(* CODESYS project core.library
   Title: CW_Core
   Version: 0.3.0
   Placeholder: CW_Core
   Company: Climeworks AG

Project tree, tasks and I/O mapping:
  libraries: Tc2_Standard, * (Beckhoff Automation GmbH); Tc2_System, * (Beckhoff Automation GmbH); Tc2_Utilities, * (Beckhoff Automation GmbH); Tc3_Module, * (Beckhoff Automation GmbH); VisuDialogs, * (System)
  Clock/
    function block FB_Clock [ST]: end_of_day, ready, toString
    interface ITF_Clock: end_of_day, ready, toString
  i18n/
    data type E_Language
    function F_GetLanguageId [ST]
    function block FB_TextList [ST]: FB_init, get
    visualisation Frame_SwitchLanguage
    data type T_TranslatableName
    data type T_TranslatableText
  Implicit/
    function F_CheckRangeSigned [ST]
    function F_CheckRangeUnsigned [ST]
  Log/
    DataLogger/
      data type E_LoggerError
      function block FB_EventLoggableLogger [ST]: collectLog, FB_init, run
      function block FB_EventLogger [ST]: updateTimeFormat, useMilliseconds, _trigger, FB_init, trigger, triggerIf, triggerWithTime, write
      function block FB_ExternalTimestamp [ST]: end_of_day, ready, reset, setTime, toString
      function block FB_TimedLoggableLogger [ST]: collectLog, FB_init, run
      function block FB_TimedLogger [ST]: FB_init, write_sampled
      interface ITF_LogDataCollector: collectLog
      data type TIMESTAMPSTRING
    Interfaces/
      interface ITF_LogExtension: getLogTrigger
      interface ITF_Loggable: toLog
      interface ITF_Recordable: enableSelectionMode
    LogStack/
      data type E_LogSequence
      function block FB_LogStackManager [ST]: available, empty, getKey, getStackLevel, nextReadData, nextWritePtr, writeToStack, writeToStackData, writeToStackHeader
      function block FB_ResponseStackManager [ST]: getResponse, storeResponse
      interface ITF_WritableStack: available, getKey, writeToStackData, writeToStackHeader
      data type ST_logStackData
      data type ST_ResponseStack
    LogString/
      function block FB_LogString [ST]: logBoolProperty, logUdintProperty, logUintProperty, logBool, logReal, logString, logUdint, logUint, append, clear, concat, getLine, length, logAny, logValue, num_lines
      data type LOGSTRING
    LogWriter/
      function block FB_LogWriter [ST]: FB_init, full_filename, handleResponse, updateFileName, updateFileType, write
      data type ST_LogMessage
    data type E_LogMode
    global variables PL_Log
  ManualRecording/
    visualisation Frame_ManualRecording_display
    data type ST_Record
  Math/
    function F_NotZero [ST]
    function F_Ramp [ST]
  Mixin/
    Fallible/
      interface ITF_Fallible: get_name, has_error
    Pressure/
      data type E_PressureUnit
      function block FB_PressureMixin [ST]: bar, display_accuracy, from_mbar, mbar, pa
  Physics/
    SteamCondition/
      function F_P_SAT [ST]
      function F_T_SAT [ST]
    function F_sim_pressureFlow [ST]
  StringSizes/
    data type NAME_STRING
    global variables PL_StringSizes
    data type TAG_STRING
  TEST/
    lib/
      function block FB_Test [ST]: check
      program TEST_TEMPLATE [ST]
    Utils/
      program TEST_BITS [ST]
      program TEST_TIMESTRUCT_INCREMENT [ST]: assertEqual
    program TEST [ST]
  Utils/
    Bits/
      function SET_BIT_IN_BYTE [ST]
      function SET_BIT_IN_BYTE_ARRAY [ST]
    Endian/
      function F_IntSwapEndian [ST]
      function F_SafeRealSwapEndian [ST]
      function F_SafeRealSwapWords [ST]
      data type Float32
      data type Int16
    Limits/
      Visu/
        visualisation Frame_IntLimits
        visualisation Frame_RealLimits
        visualisation Frame_UdintLimits
        visualisation Frame_UsintLimits
        text list TL_DisplayAccuracy
      data type ST_BaseLimits
      data type ST_DintLimits
      data type ST_IntLimits
      data type ST_RealLimits
      data type ST_UdintLimits
      data type ST_UintLimits
      data type ST_UsintLimits
    String/
      Concat/
        function CONCAT3 [ST]
        function CONCAT4 [ST]
        function CONCAT5 [ST]
        function CONCAT6 [ST]
      Placeholder/
        function F_ResolvePlaceholder [ST]
        data type PLACEHOLDER_STRING
      function F_FindAndReplace [ST]
      function F_FindAndReplaceAll [ST]
      function F_Glue [ST]
      function F_ReplaceX [ST]
      function FILL_WIDTH [ST]
    Ternary/
      function BOOL_TO_TERNARY [ST]
      data type E_Ternary
    Time/
      data type E_TIME_UNIT
      function block FB_Blinker [ST]
      function block FB_TimeDelta [ST]: reset
      function block FB_TON_PAUSABLE [ST]
      function SYSTEMTIME_TO_STRING [ST]
      function TIME_TO_FSTRING [ST]
      function TIMESTRUCT_INCREMENT [ST]
    function block FB_RememberRestore [ST]: remember, restore
    function block FB_ResourceManager [ST]: available, FB_init, release, reserve
*)

// i18n/E_Language
{attribute 'qualified_only'}
TYPE E_Language :
(
	de := 0,
	en,
	num
)UINT;
END_TYPE

// i18n/T_TranslatableName
TYPE T_TranslatableName : ARRAY[0..E_Language.num-1] OF NAME_STRING; END_TYPE

// i18n/T_TranslatableText
TYPE T_TranslatableText : ARRAY[0..E_Language.num-1] OF T_MaxString; END_TYPE

// Log/DataLogger/E_LoggerError
{attribute 'qualified_only'}
{attribute 'strict'}
TYPE E_LoggerError :
(
	ok := 0,
	trigger_overflow
) UDINT;
END_TYPE

// Log/DataLogger/TIMESTAMPSTRING
TYPE TIMESTAMPSTRING : STRING(30); END_TYPE

// Log/LogStack/E_LogSequence
{attribute 'qualified_only'}
{attribute 'strict'}
TYPE E_LogSequence :
(
	daily		:= 1,
	weekly		:= 2,
	monthly		:= 4,
	yearly		:= 8,
	perCycle	:= 16,
	unlimited	:= 32,
	other1		:= 64,
	other2		:= 128
) WORD;
END_TYPE

// Log/LogStack/ST_logStackData
TYPE ST_logStackData :
STRUCT
	type_of_data : INT;			// 0: data	1:Header
	key : INT;					// Response: Key ID
	file_name : STRING[64];		// C# Len=65		 = “Betriebsdaten.log”
	file_type : WORD;			// FileType          = 01h (=daily)
								// 1: daily
								// 2: weekly
								// 4: monthly
								// 8: yearly
								// 16: per cycle
								// 32: unlimited
								// 64: other features (example: overwrite file on restart)
								// 128: other features
	cycle : INT;				// Process Cycle when fileType 16 is used
	option : INT;
	header_or_data : STRING[255]; // C# Len=256
	eom : BOOL;					// End of Message
END_STRUCT
END_TYPE

// Log/LogStack/ST_ResponseStack
TYPE ST_ResponseStack :
STRUCT
	// Response
	key			:INT;			// Response: Key ID
	fault_code	:INT;			// NONE 				= 0	V1.00-X31
        						// KEY 					= 1 // Key ist dem Feurer-Tool nicht mehr bekannt. Vermutlich wurde es neugestartet. Header muss erneut gesendet werden.
        						// FILE_MISSING 		= 2
        						// FILENAME_MISSING 	= 3
        						// FILESYSTEM 			= 4 // Wahrscheinlich Speicher voll?
        						// SERIALIZATION 		= 5
        						// NULLMSG 				= 99
	error		:BOOL;			// Response: Error
END_STRUCT
END_TYPE

// Log/LogString/LOGSTRING
TYPE LOGSTRING : ARRAY[1..PL_Log.max_lines] OF STRING(255); END_TYPE

// Log/LogWriter/ST_LogMessage
TYPE ST_LogMessage :
STRUCT
	header	: FB_LogString := ( get_header := TRUE, force_get_data := TRUE );
	data	: FB_LogString;
END_STRUCT
END_TYPE

// Log/E_LogMode
{attribute 'qualified_only'}
TYPE E_LogMode :
(
	no := 0,
	yes,
	on_change
);
END_TYPE

// ManualRecording/ST_Record
TYPE ST_Record :
STRUCT
	enabled : BOOL;  // if true, this will be recorded in the manual recording
	selection_mode : BOOL;  // if true, this should show an option on the HMI to be selected for recording
END_STRUCT
END_TYPE

// Mixin/Pressure/E_PressureUnit
{attribute 'qualified_only'}
{attribute 'strict'}
TYPE E_PressureUnit :
(
	mbar := 0,
	bar,
	pa
);
END_TYPE

// StringSizes/NAME_STRING
TYPE NAME_STRING : STRING(PL_StringSizes.name_string_size); END_TYPE

// StringSizes/TAG_STRING
TYPE TAG_STRING : STRING(PL_StringSizes.tag_string_size); END_TYPE

// Utils/Endian/Float32
TYPE Float32 :
UNION
	float : REAL;
	dword_ : DWORD;
	words : ARRAY[0..1] OF WORD;
	bytes : ARRAY[0..3] OF BYTE;
END_UNION
END_TYPE

// Utils/Endian/Int16
TYPE Int16 :
UNION
	uinteger : UINT;
	integer : INT;
	bytes : ARRAY[0..1] OF BYTE;
END_UNION
END_TYPE

// Utils/Limits/ST_BaseLimits
TYPE ST_BaseLimits :
STRUCT
	display_font_size : UINT(0..40) := 9;  //pt
END_STRUCT
END_TYPE

// Utils/Limits/ST_DintLimits
TYPE ST_DintLimits EXTENDS ST_BaseLimits :
STRUCT
	low : DINT;
	high : DINT;
END_STRUCT
END_TYPE

// Utils/Limits/ST_IntLimits
TYPE ST_IntLimits EXTENDS ST_BaseLimits :
STRUCT
	low : INT;
	high : INT;
END_STRUCT
END_TYPE

// Utils/Limits/ST_RealLimits
TYPE ST_RealLimits EXTENDS ST_BaseLimits :
STRUCT
	low : REAL;
	high : REAL;
	display_accuracy : UINT(0..4) := 1;
END_STRUCT
END_TYPE

// Utils/Limits/ST_UdintLimits
TYPE ST_UdintLimits EXTENDS ST_BaseLimits:
STRUCT
	low : UDINT;
	high : UDINT;
END_STRUCT
END_TYPE

// Utils/Limits/ST_UintLimits
TYPE ST_UintLimits EXTENDS ST_BaseLimits :
STRUCT
	low : UINT;
	high : UINT;
END_STRUCT
END_TYPE

// Utils/Limits/ST_UsintLimits
TYPE ST_UsintLimits EXTENDS ST_BaseLimits :
STRUCT
	low : USINT;
	high : USINT;
END_STRUCT
END_TYPE

// Utils/String/Placeholder/PLACEHOLDER_STRING
TYPE PLACEHOLDER_STRING : STRING(3); END_TYPE

// Utils/Ternary/E_Ternary
{attribute 'qualified_only'}
{attribute 'strict'}
TYPE E_Ternary :
(
	unset := 0,
	yes,
	no
)USINT;
END_TYPE

// Utils/Time/E_TIME_UNIT
{attribute 'qualified_only'}
{attribute 'strict'}
TYPE E_TIME_UNIT :
(
	millisecond := 0,
	second,
	minute,
	hour,
	day
);
END_TYPE

// Log/PL_Log
{attribute 'qualified_only'}
VAR_GLOBAL CONSTANT
	max_lines : INT := 65;  // size of FB_LogString
	log_stack_size : INT := 90;  // size of Log Stack (should be bigger than log string)
END_VAR

// StringSizes/PL_StringSizes
{attribute 'qualified_only'}
VAR_GLOBAL CONSTANT
	name_string_size : UINT := 40;
	tag_string_size : UINT := 15;
END_VAR

// Clock/FB_Clock
FUNCTION_BLOCK FB_Clock IMPLEMENTS ITF_Clock
VAR_OUTPUT
	date_time_initialized	: BOOL; // TRUE, sobald dateTime korrekten Wert enthält
	date_time				: TIMESTRUCT; // Aktuelle Datumzeit des Systems
	end_of_year				: BOOL; // TRUE bei Jahreswechsel
	end_of_month			: BOOL; // TRUE bei Monatswechsel
	_end_of_day				: BOOL; // TRUE bei Tageswechsel
END_VAR
VAR
	nt_get_time				: NT_GetTime;
END_VAR
VAR PERSISTENT
	last_date_time			: TIMESTRUCT; // Zeit des letzten Zyklus
END_VAR

// Datum und Uhrzeit in einen Timestruct schreiben
nt_get_time(START:=TRUE, TIMESTR=>date_time);
IF NOT nt_get_time.BUSY THEN
	date_time_initialized := TRUE;
	nt_get_time(START:=FALSE); // Zurücksetzen
ELSIF date_time_initialized THEN
	// increment time while nt_get_time is busy to prevent duplicate timestamp in logs
	date_time := TIMESTRUCT_INCREMENT( date_time, UDINT_TO_UINT(TwinCAT_SystemInfoVarList._TaskInfo[GETCURTASKINDEXEX()].CycleTime/10000) );
END_IF

// Sobald Systemzeit gelesen wurde..
IF date_time_initialized THEN

	// Jahreswechsel detektieren
	IF (date_time.wYear > last_date_time.wYear) THEN
		end_of_year := TRUE;
	ELSE
		end_of_year := FALSE;
	END_IF

	// Monatswechsel detektieren
	IF (date_time.wMonth > last_date_time.wMonth) AND date_time.wYear = last_date_time.wYear OR (date_time.wYear > last_date_time.wYear) THEN
		end_of_month := TRUE;
	ELSE
		end_of_month := FALSE;
	END_IF

	// Mitternacht detektieren
	IF (date_time.wDay > last_date_time.wDay) AND date_time.wMonth = last_date_time.wMonth OR (date_time.wMonth > last_date_time.wMonth) THEN
		_end_of_day := TRUE;
	ELSE
		_end_of_day := FALSE;
	END_IF

	// Letztes Datum merken
	last_date_time	:= date_time;
END_IF

PROPERTY end_of_day : BOOL
GET
end_of_day := _end_of_day;
END_GET
END_PROPERTY

PROPERTY ready : BOOL
// returns true, if clock is ready for use
GET
ready := date_time_initialized;
END_GET
END_PROPERTY

METHOD toString : STRING
VAR_INPUT
	format		: STRING;
END_VAR
toString := SYSTEMTIME_TO_STRING( date_time, format );
END_METHOD

END_FUNCTION_BLOCK

// Utils/Time/TIMESTRUCT_INCREMENT
FUNCTION TIMESTRUCT_INCREMENT : TIMESTRUCT
VAR_INPUT
	base : TIMESTRUCT;
	increment : UINT;  // in ms
END_VAR

// increases the timestruct by increment
IF	base.wMilliseconds + increment < 1000 THEN
	TIMESTRUCT_INCREMENT := base;
	TIMESTRUCT_INCREMENT.wMilliseconds := base.wMilliseconds + increment;
ELSE
	// DT looses milliseconds (rounded)
	TIMESTRUCT_INCREMENT := base;
	TIMESTRUCT_INCREMENT.wMilliseconds := 0;
	TIMESTRUCT_INCREMENT := DT_TO_SYSTEMTIME(SYSTEMTIME_TO_DT(TIMESTRUCT_INCREMENT) + UINT_TO_TIME((base.wMilliseconds + increment)/1000*1000));
	TIMESTRUCT_INCREMENT.wMilliseconds := ( base.wMilliseconds + increment ) MOD 1000;
END_IF

END_FUNCTION

// Clock/ITF_Clock
INTERFACE ITF_Clock

PROPERTY end_of_day : BOOL
GET
END_GET
END_PROPERTY

PROPERTY ready : BOOL
// returns true, if clock is ready for use
GET
END_GET
END_PROPERTY

METHOD toString : STRING
VAR_INPUT
	format		: STRING;
END_VAR
END_METHOD

END_INTERFACE

// Utils/Time/SYSTEMTIME_TO_STRING
FUNCTION SYSTEMTIME_TO_STRING : STRING
VAR_INPUT
	system_time	: TIMESTRUCT;
	format		: STRING;
END_VAR
VAR
	tmp_string	: STRING;
END_VAR

SYSTEMTIME_TO_STRING := format;

// aktuelle Zeit (%T)
SYSTEMTIME_TO_STRING := F_FindAndReplace( SYSTEMTIME_TO_STRING, '%T', '%H:%M:%S' );


// Jahr 4-Stellig
IF system_time.wYear < 10 THEN
	tmp_string := CONCAT ('0', WORD_TO_STRING(system_time.wYear));
ELSE
	tmp_string := WORD_TO_STRING(system_time.wYear);
END_IF
SYSTEMTIME_TO_STRING := F_FindAndReplace( SYSTEMTIME_TO_STRING, '%Y', tmp_string );


// Monat
IF system_time.wMonth < 10 THEN
	tmp_string := CONCAT ('0', WORD_TO_STRING(system_time.wMonth));
ELSE
	tmp_string := WORD_TO_STRING(system_time.wMonth);
END_IF
SYSTEMTIME_TO_STRING := F_FindAndReplace( SYSTEMTIME_TO_STRING, '%m', tmp_string );


// Tag des Monats
IF system_time.wDay < 10 THEN
	tmp_string := CONCAT ('0', WORD_TO_STRING(system_time.wDay));
ELSE
	tmp_string := WORD_TO_STRING(system_time.wDay);
END_IF
SYSTEMTIME_TO_STRING := F_FindAndReplace( SYSTEMTIME_TO_STRING, '%d', tmp_string );


// h (%H) (Bereich 00 bis 23)
IF system_time.wHour < 10 THEN
	tmp_string := CONCAT ('0', WORD_TO_STRING(system_time.wHour));
ELSE
	tmp_string := WORD_TO_STRING(system_time.wHour);
END_IF
SYSTEMTIME_TO_STRING := F_FindAndReplace( SYSTEMTIME_TO_STRING, '%H', tmp_string );

// min (%M) (Bereich 00 bis 59)
IF system_time.wMinute < 10 THEN
	tmp_string := CONCAT ('0', WORD_TO_STRING(system_time.wMinute));
ELSE
	tmp_string := WORD_TO_STRING(system_time.wMinute);
END_IF
SYSTEMTIME_TO_STRING := F_FindAndReplace( SYSTEMTIME_TO_STRING, '%M', tmp_string );

// sec (%S)
IF system_time.wSecond < 10 THEN
	tmp_string := CONCAT ('0', WORD_TO_STRING(system_time.wSecond));
ELSE
	tmp_string := WORD_TO_STRING(system_time.wSecond);
END_IF
SYSTEMTIME_TO_STRING := F_FindAndReplace( SYSTEMTIME_TO_STRING, '%S', tmp_string );

// Millisec (%f)
IF system_time.wMilliseconds < 10 THEN
	tmp_string := CONCAT ('00', WORD_TO_STRING(system_time.wMilliseconds));
ELSIF system_time.wMilliseconds < 100 THEN
	tmp_string := CONCAT ('0', WORD_TO_STRING(system_time.wMilliseconds));
ELSE
	tmp_string := WORD_TO_STRING(system_time.wMilliseconds);
END_IF
SYSTEMTIME_TO_STRING := F_FindAndReplace( SYSTEMTIME_TO_STRING, '%f', tmp_string );

END_FUNCTION

// Utils/String/F_FindAndReplace
FUNCTION F_FindAndReplace : STRING
VAR_INPUT
	str : T_MaxString;
	find_str : T_MaxString;
	replace_str : T_MaxString;
END_VAR
VAR_OUTPUT
	found : BOOL; 
END_VAR
VAR
	p : INT;
END_VAR

p := FIND( str, find_str );
found := p > 0;
IF found THEN
	F_FindAndReplace := REPLACE( str, replace_str, LEN(find_str), p );
ELSE
	F_FindAndReplace := str;
END_IF

END_FUNCTION

// i18n/F_GetLanguageId
FUNCTION F_GetLanguageId : E_Language
// Gibt die aktuelle Sprache der Visu zurück
VAR_INPUT
END_VAR
VAR
	language : STRING;
END_VAR

language := VisuElems.cmpDynamictext.DynamicTextGetCurrentLanguage();
IF language = '' OR language = 'default' OR language = 'de' THEN
	F_GetLanguageId := E_Language.de;
ELSE
	F_GetLanguageId := E_Language.en;
END_IF

END_FUNCTION

// i18n/FB_TextList
FUNCTION_BLOCK FB_TextList
VAR_INPUT
END_VAR
VAR_OUTPUT
END_VAR
VAR
	text_list_path : STRING;
END_VAR

METHOD FB_init : BOOL
VAR_INPUT
	bInitRetains : BOOL; // if TRUE, the retain variables are initialized (warm start / cold start)
	bInCopyCode   : BOOL;  // if TRUE, the instance afterwards gets moved into the copy code (online change)
	text_list : STRING;
END_VAR
text_list_path := text_list;
END_METHOD

METHOD get : STRING
VAR_INPUT
	index : UINT;
END_VAR
VAR
	language : STRING;
	index_string : STRING;
END_VAR
index_string := UINT_TO_STRING(index);

language := VisuElems.cmpDynamictext.DynamicTextGetCurrentLanguage();
IF language = '' OR language = 'default' THEN
	get := VisuElems.cmpDynamictext.DynamicTextGetDefaultText(ADR(text_list_path), ADR(index_string))^;
ELSE
	get := VisuElems.cmpDynamictext.DynamicTextGetText(ADR(text_list_path), ADR(index_string))^;
END_IF
END_METHOD

END_FUNCTION_BLOCK

// Implicit/F_CheckRangeSigned
// Implicitly generated code : DO NOT EDIT
FUNCTION F_CheckRangeSigned : DINT
VAR_INPUT
	value, lower, upper: DINT;
END_VAR

// Implicitly generated code : Only an Implementation suggestion
{noflow}
IF (value < lower) THEN
	F_CheckRangeSigned := lower;
ELSIF(value > upper) THEN
	F_CheckRangeSigned := upper;
ELSE
	F_CheckRangeSigned := value;
END_IF
{flow}

END_FUNCTION

// Implicit/F_CheckRangeUnsigned
// Implicitly generated code : DO NOT EDIT
FUNCTION F_CheckRangeUnsigned : UDINT
VAR_INPUT
	value, lower, upper: UDINT;
END_VAR

// Implicitly generated code : Only an Implementation suggestion
{noflow}
IF (value < lower) THEN
	F_CheckRangeUnsigned := lower;
ELSIF(value > upper) THEN
	F_CheckRangeUnsigned := upper;
ELSE
	F_CheckRangeUnsigned := value;
END_IF
{flow}

END_FUNCTION

// Log/DataLogger/FB_EventLoggableLogger
FUNCTION_BLOCK FB_EventLoggableLogger EXTENDS FB_EventLogger IMPLEMENTS ITF_LogDataCollector
VAR
	// loggable to get data from
	loggable : ITF_Loggable;

	// settings
	log_type : UINT;
END_VAR

METHOD collectLog : BOOL
VAR_IN_OUT
	log_string	: FB_LogString;
END_VAR
VAR_INPUT
	timestamp : TIMESTAMPSTRING;  // is "Time;" for header and current timestamp + ';' as string for data
END_VAR
log_string.append(timestamp);
loggable.toLog( log_string, log_type );
END_METHOD

METHOD FB_init : BOOL
VAR_INPUT
	bInitRetains : BOOL; // if TRUE, the retain variables are initialized (warm start / cold start)
	bInCopyCode : BOOL;  // if TRUE, the instance afterwards gets moved into the copy code (online change)
	file_name	: STRING(53);
END_VAR
log_writer.updateFileName(file_name);
END_METHOD

METHOD run : BOOL
VAR_INPUT
	loggable : ITF_Loggable;
	stack : ITF_WritableStack;
	clock : ITF_Clock;
	file_writer_connected : BOOL;
END_VAR
// Den loggable für die collect-Methoden erreichbar machen
THIS^.loggable := loggable;
// Logger laufen lassen.
write( data_collector := THIS^, stack, file_writer_connected );
END_METHOD

END_FUNCTION_BLOCK

// Log/DataLogger/FB_EventLogger
FUNCTION_BLOCK FB_EventLogger;
VAR_INPUT
	force_get_data : BOOL; //TRUE: force the values of all elements to be appended to the log_string, FALSE: elements decide if append the data or not
END_VAR
VAR_OUTPUT
	error : BOOL;
	error_id : UDINT;
	last_timestamp : TIMESTAMPSTRING;  // last timestamp of an internal trigger to be used to inform external triggers
END_VAR
VAR_INPUT
	max_triggering_interval : USINT := 3; // Maximum interval between consecutive triggering (i.e. lines in the log file). Unit is program cycles
END_VAR
VAR
	message : ST_LogMessage;
	header_cached : BOOL;  // TRUE, wenn header gecached wurde
	// triggering
	triggered : BOOL; // TRUE: event logger has been triggered, FALSE: event logger is not being triggered

	// writer
	log_writer : FB_LogWriter('EventLogger', E_LogSequence.daily);
	data_collected : BOOL; // TRUE: data has been collected

	// timestamp settings
	time_header : TIMESTAMPSTRING := 'Time;';
	time_format : STRING := '%Y-%m-%d %H:%M:%S';
	timestamp : TIMESTAMPSTRING;
END_VAR

METHOD updateTimeFormat : BOOL
VAR_INPUT
	new_time_format : STRING;
END_VAR
time_format := new_time_format;
END_METHOD

METHOD useMilliseconds : BOOL
VAR_INPUT
	use_milliseconds : BOOL;
END_VAR
IF use_milliseconds THEN
	time_format := CONCAT( time_format, '.%f' );
END_IF
END_METHOD

// basic trigger
METHOD PRIVATE _trigger : BOOL
VAR_INPUT
	clock : ITF_Clock;
END_VAR
{warning 'the clock may not be ready here. check somewhere else'}
timestamp := clock.toString(time_format);
triggered := TRUE;
END_METHOD

METHOD FB_init : BOOL
VAR_INPUT
	bInitRetains : BOOL; // if TRUE, the retain variables are initialized (warm start / cold start)
	bInCopyCode : BOOL;  // if TRUE, the instance afterwards gets moved into the copy code (online change)
END_VAR
log_writer.updateFileType(E_LogSequence.daily);  // legacy default.
END_METHOD

// trigger for module internal triggering with own timestamp
METHOD trigger : BOOL
VAR_INPUT
	clock : ITF_Clock;
END_VAR
{warning 'the clock may not be ready here. check somewhere else'}
_trigger(clock);
last_timestamp := timestamp;  // remember for external trigger
END_METHOD

METHOD triggerIf : BOOL
VAR_INPUT
	condition : BOOL;
	clock : ITF_Clock;
END_VAR
IF condition THEN
	trigger(clock);
END_IF
triggerIf := triggered;
END_METHOD

// trigger for external triggering with other timestamp
METHOD triggerWithTime : BOOL
VAR_INPUT
	external_timestamp : REFERENCE TO FB_ExternalTimestamp;
END_VAR
IF external_timestamp.triggered THEN
	_trigger(external_timestamp);
END_IF
END_METHOD

METHOD write : BOOL
VAR_INPUT
	data_collector : ITF_LogDataCollector;
	stack : ITF_WritableStack;
	file_writer_connected : BOOL;
END_VAR
VAR_INST
	write_to_log : BOOL;
	consecutive_trigger_counter : USINT;
END_VAR
// 1. Header zusammensetzen und senden
IF NOT header_cached THEN
	message.header.clear();
	data_collector.collectLog( message.header, time_header );
	header_cached := TRUE;
	write_to_log := TRUE;
END_IF

// 2. If log_writer has not been initialized, i.e. header has not been written, force get a complete log_string of data (second line after header should always been complete).
IF NOT log_writer.status_initialized THEN
	message.data.force_get_data := TRUE;
ELSE
	message.data.force_get_data := force_get_data;
END_IF

// Trigger overflow watchdog
IF triggered THEN
	consecutive_trigger_counter := consecutive_trigger_counter + 1;

	IF consecutive_trigger_counter > max_triggering_interval THEN
		error := TRUE;
		error_id := E_LoggerError.trigger_overflow;
		consecutive_trigger_counter := 0;
		data_collected := FALSE;
	END_IF
ELSE
	error := FALSE;
	consecutive_trigger_counter := 0;
	data_collected := FALSE;
END_IF

// 2. Daten zusammensetzen
IF triggered AND NOT data_collected THEN
	message.data.clear();
	data_collector.collectLog( message.data, CONCAT(timestamp, ';') );
	data_collected := TRUE; // reset
END_IF
triggered := FALSE;

// 4. Header und/oder Daten schreiben
// TODO: Auslesen, ob ein Fehler aufgetreten ist #SafetyChecks
// IMPORTANT: this write method must be called regularly, to resend the header if pydialogs restarted
IF log_writer.write(message, stack, file_writer_connected) THEN
	message.data.clear();
END_IF

// Reset Error ID
IF NOT error THEN
	error_id := E_LoggerError.ok;
END_IF
END_METHOD

END_FUNCTION_BLOCK

// Log/LogWriter/FB_LogWriter
FUNCTION_BLOCK FB_LogWriter
VAR_INPUT
	cycle : INT;  // Process Cycle when fileType "perCycle" is used
END_VAR
VAR_OUTPUT
	// TODO: Bei error könnte eine Warnung auslösen.
	error_response :BOOL;
	fault_code :INT;			// NONE 				= 0	V1.00-X31
        						// KEY 					= 1 // Key ist dem Feurer-Tool nicht mehr bekannt. Vermutlich wurde es neugestartet. Header muss erneut gesendet werden.
        						// FILE_MISSING 		= 2
        						// FILENAME_MISSING 	= 3
        						// FILESYSTEM 			= 4 // Wahrscheinlich Speicher voll?
        						// SERIALIZATION 		= 5
        						// NULLMSG 				= 99
	error_full_stack : BOOL;
	status_initialized : BOOL := FALSE;
END_VAR
VAR
	// settings
	key : INT;  // Response: Key ID
	file_prefix : STRING(20);
	file_extension : STRING(10) := 'csv';
	file_name : STRING(60);  // Dateiname ohne Endung
	file_type : E_LogSequence;  // FileType

	//
	//stack_manager : REFERENCE TO FB_LogStackManager;
END_VAR

METHOD FB_init : BOOL
VAR_INPUT
	bInitRetains : BOOL; // if TRUE, the retain variables are initialized (warm start / cold start)
	bInCopyCode : BOOL;  // if TRUE, the instance afterwards gets moved into the copy code (online change)
	file_name	: STRING(53);
	file_type	: E_LogSequence; // FileType
END_VAR
THIS^.file_name := file_name;
THIS^.file_type := file_type;
END_METHOD

PROPERTY full_filename : STRING(100)
GET
IF file_prefix <> '' THEN
	full_filename := CONCAT5(file_prefix, '_', file_name, '.', file_extension);
ELSE
	full_filename := CONCAT3(file_name, '.', file_extension);
END_IF
END_GET
END_PROPERTY

METHOD handleResponse : BOOL
VAR_INPUT
	response : ST_ResponseStack;
END_VAR
error_response := response.error;
fault_code := response.fault_code;
END_METHOD

METHOD updateFileName : BOOL
VAR_INPUT
	new_file_name : STRING(60);
END_VAR
file_name := new_file_name;
status_initialized := FALSE; // Muss neu initialisiert werden.
END_METHOD

METHOD updateFileType : BOOL
VAR_INPUT
	new_file_type : E_LogSequence;
END_VAR
file_type := new_file_type;
status_initialized := FALSE; // Muss neu initialisiert werden.
END_METHOD

METHOD write : BOOL
VAR_IN_OUT
	message	: ST_LogMessage;
END_VAR
VAR_INPUT
	stack_manager : ITF_WritableStack;
	file_writer_connected : BOOL;
END_VAR
VAR
	i : UINT;
END_VAR
VAR_INST
	initialized: BOOL;
END_VAR
// get key the first time
IF NOT initialized THEN
	key := stack_manager.getKey();
	initialized := TRUE;
END_IF

// Filing anhalten, wenn Dialogs nicht verbunden ist.
IF NOT file_writer_connected THEN
	status_initialized := FALSE; // Header muss erneut geschrieben werden, wenn Verbindung wieder aufgebaut wurde.
	RETURN;
END_IF

// Header nach Fehler erneut senden.
IF error_response OR fault_code <> 0 THEN
	status_initialized := FALSE;
END_IF

// Header
IF NOT status_initialized AND message.header.length > 0 AND stack_manager.available >= message.header.num_lines THEN
	// Setup & Init
	FOR i:=1 TO message.header.num_lines DO
		// Teil i Header in den Stack schreiben
		error_full_stack := NOT stack_manager.writeToStackHeader (
			key := key,
			file_name := full_filename,
			file_type := file_type,  // FileType
			cycle := cycle,  // Process Cycle when fileType 16 is used
			option := 0,
			header := message.header.getLine(i),  // C# Len=256
			eom := (i=message.header.num_lines)  // End of Message
		);
	END_FOR
	status_initialized:=TRUE;
END_IF

// Data
IF status_initialized AND message.data.length > 0 AND stack_manager.available >= message.data.num_lines THEN
	FOR i:=1 TO message.data.num_lines DO
		// Hier werden die Daten in den Stack geschrieben
		error_full_stack := NOT stack_manager.writeToStackData(
			key := key,
			data := message.data.getLine(i),
			eom := (i=message.data.num_lines)  // End of Message
		);
	END_FOR
	write := TRUE;
END_IF
END_METHOD

END_FUNCTION_BLOCK

// Log/LogStack/FB_LogStackManager
{attribute 'analysis' := '-2'} // yes this is empty
FUNCTION_BLOCK FB_LogStackManager IMPLEMENTS ITF_WritableStack
VAR
	log_stack_read				:INT := 0;
	log_stack_write				:INT := 0;
	log_stack_data				:ARRAY[0..PL_Log.log_stack_size-1] OF ST_logStackData;
	stack_full					:BOOL;
	//log_stack_sent, log_stack_received :ARRAY[0..log_stack_size-1] OF BOOL;
	
	next_key : INT;
END_VAR

PROPERTY available : UINT
GET
available := INT_TO_UINT(( log_stack_read - log_stack_write - 1 + PL_Log.log_stack_size ) MOD PL_Log.log_stack_size);
END_GET
END_PROPERTY

PROPERTY empty : BOOL
GET
empty := log_stack_read = log_stack_write;
END_GET
END_PROPERTY

METHOD getKey : INT;
// Do not call this method in declaration part of in FB_init
getKey := next_key;
next_key := next_key + 1;
END_METHOD

METHOD getStackLevel : REAL
VAR_INPUT
END_VAR
getStackLevel := INT_TO_REAL( ( log_stack_write - log_stack_read + PL_Log.log_stack_size ) MOD PL_Log.log_stack_size ) / PL_Log.log_stack_size;
END_METHOD

METHOD nextReadData : ST_logStackData // Gibt Referenz auf nächte zu lesende Zeile zurück.
VAR_INPUT
END_VAR
log_stack_read := (log_stack_read + 1) MOD PL_Log.log_stack_size;
nextReadData := log_stack_data[log_stack_read];
END_METHOD

METHOD PRIVATE nextWritePtr : POINTER TO ST_logStackData // Gibt Pointer auf nächte zu lesende Zeile zurück.
VAR_INPUT
END_VAR
VAR
	tmp : INT;
END_VAR
tmp := (log_stack_write + 1) MOD PL_Log.log_stack_size;

// Wenn Stack voll ist, keine Referenz zurückgeben. Write-Pointer bleibt unverändert.
IF stack_full := tmp = log_stack_read THEN
	nextWritePtr := 0;
	//Setze EOM beim letzen Eintrag
	log_stack_data[log_stack_write].eom := TRUE;
	RETURN;
END_IF
log_stack_write := tmp;

nextWritePtr := ADR(log_stack_data[log_stack_write]);
END_METHOD

METHOD PRIVATE writeToStack : BOOL // Gibt True zurück, wenn In Stack geschrieben werden konnte.
VAR_INPUT
	type_of_data		:INT;			// Header = 0, Data = 1
	key			:INT;			// Response: Key ID
	file_name 		:STRING[64];	// C# Len=65		 = “Betriebsdaten.log”
	file_type		:WORD;			// FileType          = 01h (=daily)
	cycle			:INT;			// Process Cycle when fileType 16 is used
	option			:INT;
	header_or_data	:STRING[255];	// C# Len=256
	eom				:BOOL;			// End of Message
END_VAR
VAR
	write		: POINTER TO ST_logStackData;
END_VAR
write := nextWritePtr();
IF write <> 0 THEN
	write^.type_of_data := type_of_data;
	write^.key := key;
	write^.file_name := file_name;
	write^.file_type := file_type;

	write^.cycle := cycle;
	write^.option := option;
	write^.header_or_data := header_or_data;
	write^.eom := eom;
	writeToStack := TRUE; // Return TRUE
END_IF;
END_METHOD

METHOD writeToStackData : BOOL
VAR_INPUT
	key :INT;			// Response: Key ID
	data :STRING[255];	// C# Len=256
	eom :BOOL;			// End of Message
END_VAR
VAR
	success			: BOOL;
END_VAR
success := writeToStack(
	type_of_data := 1,  // Explizit data
	key := key,
	file_name := '',
	file_type := 0,
	cycle := 0,
	option := 0,
	header_or_data := data,
	eom := eom
);

writeToStackData := success;
END_METHOD

METHOD writeToStackHeader : BOOL
VAR_INPUT
	key			: INT;			// Response: Key ID
	file_name 	: STRING[64];	// C# Len=65		 = “Betriebsdaten.log”
	file_type	: E_LogSequence;	// FileType
	cycle		: INT;			// Process Cycle when fileType 16 is used
	option		: INT;
	header		: STRING[255];	// C# Len=256
	eom			: BOOL;			// End of Message
END_VAR
VAR
	success		: BOOL;
END_VAR
success := writeToStack(
	type_of_data := 0, // Explizit header
	key := key,
	file_name := file_name,
	file_type := file_type,
	cycle := cycle,
	option := option,
	header_or_data := header,
	eom := eom
);

writeToStackHeader := success;
END_METHOD

END_FUNCTION_BLOCK

// Log/LogStack/ITF_WritableStack
INTERFACE ITF_WritableStack

PROPERTY available : UINT
GET
END_GET
END_PROPERTY

METHOD getKey : INT;
END_METHOD

METHOD writeToStackData : BOOL
VAR_INPUT
	key :INT;			// Response: Key ID
	data :STRING[255];	// C# Len=256
	eom :BOOL;			// End of Message
END_VAR
END_METHOD

METHOD writeToStackHeader : BOOL
VAR_INPUT
	key			: INT;			// Response: Key ID
	file_name 	: STRING[64];	// C# Len=65		 = “Betriebsdaten.log”
	file_type	: E_LogSequence;	// FileType
	cycle		: INT;			// Process Cycle when fileType 16 is used
	option		: INT;
	header		: STRING[255];	// C# Len=256
	eom			: BOOL;			// End of Message
END_VAR
END_METHOD

END_INTERFACE

// Utils/String/Concat/CONCAT5
FUNCTION CONCAT5 : T_MaxString
VAR_INPUT
	string1 : T_MaxString;
	string2 : T_MaxString;
	string3 : T_MaxString;
	string4 : T_MaxString;
	string5 : T_MaxString;
END_VAR
VAR
END_VAR

CONCAT5 := CONCAT( CONCAT( CONCAT ( CONCAT ( string1, string2 ), string3) , string4 ), string5 );

END_FUNCTION

// Utils/String/Concat/CONCAT3
FUNCTION CONCAT3 : T_MaxString
VAR_INPUT
	string1 : T_MaxString;
	string2 : T_MaxString;
	string3 : T_MaxString;
END_VAR
VAR
END_VAR

CONCAT3 := CONCAT ( CONCAT ( string1, string2 ), string3);

END_FUNCTION

// Log/DataLogger/FB_ExternalTimestamp
// If logger is triggered with a specific timestamp (triggerWithTime), 
// this "Clock" will be used to generate the log which just returns the time that was used to trigger
FUNCTION_BLOCK FB_ExternalTimestamp IMPLEMENTS ITF_Clock
VAR_OUTPUT
	triggered : BOOL;
END_VAR
VAR
	external_time : TIMESTAMPSTRING;
END_VAR

PROPERTY end_of_day : BOOL
GET
// I wish today would never end
end_of_day := FALSE;
END_GET
END_PROPERTY

PROPERTY ready : BOOL
// returns true, if clock is ready for use
GET
// ready if an external time is set
ready := external_time <> '';
END_GET
END_PROPERTY

METHOD reset : BOOL
external_time := '';
END_METHOD

METHOD setTime : BOOL
VAR_INPUT
	timestamp : TIMESTAMPSTRING;
END_VAR
VAR_INST
	last_timestamp : TIMESTAMPSTRING;
END_VAR
// set new timestamp
external_time := timestamp;

// trigger, if timestamp changed
triggered := last_timestamp <> timestamp;  // not comparing to external_time, because that will be reset
last_timestamp := timestamp;
END_METHOD

METHOD toString : STRING
VAR_INPUT
	format		: STRING;
END_VAR
toString := external_time;
END_METHOD

END_FUNCTION_BLOCK

// Log/DataLogger/ITF_LogDataCollector
INTERFACE ITF_LogDataCollector

METHOD collectLog : BOOL
VAR_IN_OUT
	log_string : FB_LogString;
END_VAR
VAR_INPUT
	timestamp : TIMESTAMPSTRING;  // is "Time;" for header and current timestamp + ';' as string for data
END_VAR
END_METHOD

END_INTERFACE

// Log/LogString/FB_LogString
FUNCTION_BLOCK FB_LogString
VAR_INPUT
	force_get_data : BOOL := FALSE; // Force all element to return data
END_VAR
VAR_OUTPUT
	log_string	: LOGSTRING;
	overflow	: BOOL;
	get_header	: BOOL; // Gibt an, dass der Logstring den Header sammeln will statt die Daten.
END_VAR
VAR
	line : UINT(1..INT_TO_UINT(PL_Log.max_lines));
	char : UINT(0..255);
END_VAR
VAR CONSTANT
	log_string_length	: UINT := 255;
	none_value 			: STRING(1) := '';
END_VAR

{attribute 'obsolete' := 'Use logBool instead'}
METHOD logBoolProperty : BOOL
VAR_INPUT
	header 	: STRING(log_string_length); // Title von Spalte
	value	: BOOL;
END_VAR
logBoolProperty := logBoolProperty := logBool( header, value );
END_METHOD

{attribute 'obsolete' := 'Use logUdint instead'}
METHOD logUdintProperty : BOOL
VAR_INPUT
	header 	: STRING(log_string_length); // Title von Spalte
	value	: UDINT;
END_VAR
logUdintProperty := logUdint( header, value );
END_METHOD

{attribute 'obsolete' := 'Use logUint instead'}
METHOD logUintProperty : BOOL
VAR_INPUT
	header 	: STRING(log_string_length); // Title von Spalte
	value	: UINT;
END_VAR
logUintProperty := logUint( header, value );
END_METHOD

METHOD logBool : BOOL
VAR_INPUT
	header 	: STRING(log_string_length); // Title von Spalte
	value	: BOOL;
END_VAR
logValue( header, '', value );
END_METHOD

METHOD logReal : BOOL
// Loggt "value" mit Titel "sHeader".
VAR_INPUT
	header 	: STRING(log_string_length); // Title von Spalte
	unit		: STRING(10);
	value		: ANY_REAL; // Wert zu loggen (REAL oder LREAL)
	accuracy	: UINT;
END_VAR
logReal := logAny( header, unit, value, accuracy );
END_METHOD

METHOD logString : BOOL
VAR_INPUT
	header : STRING(log_string_length); // Title of column
	unit : STRING(10);
	value : STRING;
END_VAR
logString := logValue( header, unit, value );
END_METHOD

METHOD logUdint : BOOL
VAR_INPUT
	header 	: STRING(log_string_length); // Title von Spalte
	value	: UDINT;
END_VAR
logValue( header, '', value );
END_METHOD

METHOD logUint : BOOL
VAR_INPUT
	header 	: STRING(log_string_length); // Title von Spalte
	value	: UINT;
END_VAR
logValue( header, '', value );
END_METHOD

METHOD append : BOOL
// fügt dem Logstring einen String hinzu
// return: FALSE, wenn Logstring nun voll ist, sonst TRUE.
VAR_INPUT
	str : STRING(log_string_length);
END_VAR
// Ganzen String anfügen, wenn nicht zu lang
IF log_string_length-char+1 > INT_TO_UINT( LEN(str) ) THEN
	log_string[ line ] := Tc2_Standard.CONCAT( log_string[ line ], str);
	char := char + INT_TO_UINT( LEN(str) );
ELSE
	//Schreibe in diese Zeile was passt
	log_string[ line ] := Tc2_Standard.CONCAT( log_string[ line ], LEFT(str, UINT_TO_INT(log_string_length-char+1)) );
	//Fehler, wenn zu wenig Platz für String
	IF line >= INT_TO_UINT(PL_Log.max_lines) THEN
		(*
		// In Systemlog erfassen
		IF NOT overflow THEN //Nur einmal loggen
		system_logger.error(Tc2_Standard.CONCAT('Overflow: FB_LogString braucht mehr Zeilen. LOG_MAX_STRING in GlobalConst_Filing muss erhöht werden. Bisher: ', INT_TO_STRING(PL_LogString.max_lines)));
		END_IF
		*)
		overflow := TRUE;
	ELSE
		// Ansonsten, wenn es noch platz hat, gehe zur nächsten Zeile.
		line := line + 1;
		//Der Rest passt garaniert in die nächste Zeile
		log_string[ line ] := DELETE(str, UINT_TO_INT(log_string_length-char+1), 0);
		char := INT_TO_UINT( LEN(log_string[ line ]) );
	END_IF
END_IF

// return TRUE
append := NOT overflow;
END_METHOD

METHOD clear : BOOL
// Leert den Logstring
VAR_INPUT
END_VAR
VAR
	i : UINT;
END_VAR
// String leeren
FOR i:= 1 TO INT_TO_UINT(PL_Log.max_lines) DO
	log_string[i] := '';
END_FOR

// Zeiger zurücksetzen
line := 1;
char := 0;

// Fehler zurücksetzen
overflow := FALSE;
END_METHOD

METHOD concat : BOOL
// fügt die Inhalte zweier LogStrings zusammen
VAR_IN_OUT
	other_log_string : FB_LogString;
END_VAR
VAR
	i : UINT;
END_VAR
// Alle Zeilen des anderen Logstrings hinzufügen
FOR i:= 1 TO other_log_string.num_lines DO
	append( other_log_string.getLine(i) );
END_FOR
END_METHOD

METHOD getLine : STRING(255)
VAR_INPUT
	line : UINT;
END_VAR
getLine := log_string[ line ];
END_METHOD

PROPERTY length : UINT
GET
length := (line-1)*log_string_length + char;
END_GET
END_PROPERTY

METHOD PRIVATE logAny : BOOL
// Loggt "value" mit Titel "sHeader".
VAR_INPUT
	header 	: STRING(log_string_length); // Title von Spalte
	unit		: STRING(10);
	value		: __SYSTEM.AnyType; // zu loggender Wert // Kann nicht ANY sein, da sonst ANY als ANY übergeben wird und der Typ nicht erkannt wird.
	accuracy	: UINT := 2;
END_VAR
VAR
	Y 			: DINT;
	tmp_time	: DWORD;

	p_real		: POINTER TO REAL;
	p_dword 	: POINTER TO DWORD;
	p_bool		: POINTER TO BOOL;
	p_word		: POINTER TO WORD;
	p_lword		: POINTER TO LWORD;
	p_sint		: POINTER TO SINT;
	p_int		: POINTER TO INT;
	p_lint 		: POINTER TO LINT;
	p_dint		: POINTER TO DINT;
	p_usint		: POINTER TO USINT;
	p_uint		: POINTER TO UINT;
	p_udint		: POINTER TO UDINT;
	p_ulint		: POINTER TO ULINT;
	p_lreal		: POINTER TO LREAL;
	p_string	: POINTER TO STRING;
END_VAR
VAR CONSTANT
	max_size_log_value	: UINT := 50; // !!! Werte, die länger sind, werden nicht geloggt !!!
END_VAR
IF get_header THEN
	// Titel schreiben
	IF unit <> '' THEN
		append( CONCAT5( header, ' [' , unit , ']' , ';' ) );
	ELSE
		append( Tc2_Standard.CONCAT( header, ';' ) );
	END_IF
ELSE

	// Schreibt "value" Wert im logString
	//CASE value.TypeClass OF
		IF value.TypeClass = __SYSTEM.TYPE_CLASS.TYPE_BOOL THEN //BOOL
			p_bool := value.pValue;
			append(  Tc2_Standard.CONCAT( INT_TO_STRING(BOOL_TO_INT(p_bool^)), ';' ) );

		ELSIF value.TypeClass = __SYSTEM.TYPE_CLASS.TYPE_WORD THEN // WORD
			p_word := value.pValue;
			append(  Tc2_Standard.CONCAT( WORD_TO_STRING(p_word^), ';' ) );

		ELSIF value.TypeClass = __SYSTEM.TYPE_CLASS.TYPE_DWORD THEN // DWORD
			p_dword := value.pValue;
			append(  Tc2_Standard.CONCAT( DWORD_TO_STRING(p_dword^), ';' ) );

		ELSIF value.TypeClass = __SYSTEM.TYPE_CLASS.TYPE_LWORD THEN // LWORD
			p_lword := value.pValue;
			append(  Tc2_Standard.CONCAT( LWORD_TO_STRING(p_lword^), ';' ) );

		ELSIF value.TypeClass = __SYSTEM.TYPE_CLASS.TYPE_SINT THEN //SINT
			p_sint := value.pValue;
			append(  Tc2_Standard.CONCAT( SINT_TO_STRING(p_sint^), ';' ) );

		ELSIF value.TypeClass = __SYSTEM.TYPE_CLASS.TYPE_INT OR  value.TypeClass = __SYSTEM.TYPE_CLASS.TYPE_ENUM THEN// INT, ENUM
			p_int := value.pValue;
			append(  Tc2_Standard.CONCAT( INT_TO_STRING(p_int^), ';' ) );

		ELSIF value.TypeClass = __SYSTEM.TYPE_CLASS.TYPE_DINT THEN // DINT
			p_dint := value.pValue;
			append(  Tc2_Standard.CONCAT( DINT_TO_STRING(p_dint^), ';' ) );

		ELSIF value.TypeClass = __SYSTEM.TYPE_CLASS.TYPE_LINT THEN // LINT
			p_lint := value.pValue;
			append(  Tc2_Standard.CONCAT( LINT_TO_STRING(p_lint^), ';' ) );

		ELSIF value.TypeClass = __SYSTEM.TYPE_CLASS.TYPE_USINT THEN // USINT
			p_usint := value.pValue;
			append(  Tc2_Standard.CONCAT( USINT_TO_STRING(p_usint^), ';' ) );

		ELSIF value.TypeClass = __SYSTEM.TYPE_CLASS.TYPE_UINT THEN  // UINT
			p_uint := value.pValue;
			append(  Tc2_Standard.CONCAT( UINT_TO_STRING(p_uint^), ';' ) );

		ELSIF value.TypeClass = __SYSTEM.TYPE_CLASS.TYPE_UDINT THEN  // UDINT
			p_udint := value.pValue;
			append(  Tc2_Standard.CONCAT( UDINT_TO_STRING(p_udint^), ';' ) );

		ELSIF value.TypeClass = __SYSTEM.TYPE_CLASS.TYPE_ULINT THEN  // ULINT
			p_ulint := value.pValue;
			append(  Tc2_Standard.CONCAT( ULINT_TO_STRING(p_ulint^), ';' ) );

		ELSIF value.TypeClass = __SYSTEM.TYPE_CLASS.TYPE_REAL OR value.TypeClass = __SYSTEM.TYPE_CLASS.TYPE_ANYREAL THEN  // REAL, ANYREAL
			p_real := value.pValue;
			append(  Tc2_Standard.CONCAT( LREAL_TO_FMTSTR(p_real^ , UINT_TO_INT(accuracy) , TRUE ), ';' ) );

		ELSIF value.TypeClass = __SYSTEM.TYPE_CLASS.TYPE_LREAL THEN  // LREAL
			p_lreal := value.pValue;
			append(  Tc2_Standard.CONCAT( LREAL_TO_FMTSTR(p_lreal^, UINT_TO_INT(accuracy) , TRUE), ';' ) );

		ELSIF value.TypeClass = __SYSTEM.TYPE_CLASS.TYPE_STRING THEN  // STRING
			p_string := value.pValue;
			append(  Tc2_Standard.CONCAT( p_string^, ';' ) );

		ELSIF value.TypeClass = __SYSTEM.TYPE_CLASS.TYPE_TIME THEN  // TIME
			p_dword := value.pValue;
			IF unit = 's' THEN
					tmp_time := p_dword^ / 1000;
			ELSIF unit = 'min' THEN
					tmp_time := p_dword^ / 60000;
			ELSIF unit = 'h' THEN
					tmp_time := p_dword^ / 360000;
			END_IF
			append(  Tc2_Standard.CONCAT( DWORD_TO_STRING(tmp_time), ';' ) );

		ELSIF value.TypeClass = __SYSTEM.TYPE_CLASS.TYPE_DATE THEN  // DATE
			p_dword := value.pValue;
			append(  Tc2_Standard.CONCAT( DELETE( DATE_TO_STRING (DWORD_TO_DATE( p_dword^ )), 2, 1 ), ';' ) );

		ELSIF value.TypeClass = __SYSTEM.TYPE_CLASS.TYPE_TIMEOFDAY THEN  // TIMEOFDAY
			p_dword := value.pValue;
			append(  Tc2_Standard.CONCAT( DELETE( TOD_TO_STRING (DWORD_TO_TOD( p_dword^ )), 4, 1 ), ';' ) );

		ELSIF value.TypeClass = __SYSTEM.TYPE_CLASS.TYPE_DATEANDTIME THEN  // DATEANDTIME
			p_dword := value.pValue;
			append(  Tc2_Standard.CONCAT( DELETE( DT_TO_STRING (DWORD_TO_DT( p_dword^ )), 3, 1 ), ';' ) );
		END_IF
END_IF
END_METHOD

METHOD logValue : BOOL
// Loggt "value" mit Titel "sHeader".
VAR_INPUT
	header 	: STRING(log_string_length); // Title von Spalte
	unit		: STRING(10);
	value		: ANY; // Wert zu loggen (Variablenart nicht wichtig)
END_VAR
logValue := logAny( header, unit, value, 2 );
END_METHOD

PROPERTY num_lines : UINT
GET
num_lines := line;
END_GET
END_PROPERTY

END_FUNCTION_BLOCK

// Log/Interfaces/ITF_Loggable
INTERFACE ITF_Loggable EXTENDS __SYSTEM.IQueryInterface

METHOD toLog : BOOL
VAR_IN_OUT
	log_string : FB_LogString;
END_VAR
VAR_INPUT
	mode : UINT; // Legt fest, wofür LogString erzeugt werden soll
END_VAR
END_METHOD

END_INTERFACE

// Log/DataLogger/FB_TimedLoggableLogger
FUNCTION_BLOCK FB_TimedLoggableLogger EXTENDS FB_TimedLogger IMPLEMENTS ITF_LogDataCollector
VAR
	// loggable to get data from
	loggable : ITF_Loggable;

	// settings
	log_type : UINT;
END_VAR

METHOD collectLog : BOOL
VAR_IN_OUT
	log_string	: FB_LogString;
END_VAR
VAR_INPUT
	timestamp : TIMESTAMPSTRING;  // is "Time;" for header and current timestamp + ';' as string for data
END_VAR
log_string.append(timestamp);
loggable.toLog( log_string, log_type );
END_METHOD

METHOD FB_init : BOOL
VAR_INPUT
	bInitRetains : BOOL; // if TRUE, the retain variables are initialized (warm start / cold start)
	bInCopyCode : BOOL;  // if TRUE, the instance afterwards gets moved into the copy code (online change)
	sample_rate	: TIME;
	file_name	: STRING(53);
END_VAR
log_writer.updateFileName(file_name);
END_METHOD

METHOD run : BOOL
VAR_INPUT
	loggable : ITF_Loggable;
	stack : ITF_WritableStack;
	clock : ITF_Clock;
	file_writer_connected : BOOL;
END_VAR
// Den loggable für die collect-Methoden erreichbar machen
THIS^.loggable := loggable;
// Logger laufen lassen.
write_sampled( data_collector := THIS^, stack, clock, file_writer_connected );
END_METHOD

END_FUNCTION_BLOCK

// Log/DataLogger/FB_TimedLogger
FUNCTION_BLOCK FB_TimedLogger EXTENDS FB_EventLogger;
VAR
	// Sampling timer
	log_timer	: TON;
	sample_rate	: TIME := T#3S;
END_VAR

METHOD FB_init : BOOL
VAR_INPUT
	bInitRetains : BOOL; // if TRUE, the retain variables are initialized (warm start / cold start)
	bInCopyCode : BOOL;  // if TRUE, the instance afterwards gets moved into the copy code (online change)
	sample_rate	: TIME;
END_VAR
THIS^.sample_rate := sample_rate;
force_get_data := TRUE;
END_METHOD

METHOD write_sampled : BOOL
VAR_INPUT
	data_collector : ITF_LogDataCollector;
	stack : ITF_WritableStack;
	clock : ITF_Clock;
	file_writer_connected : BOOL;
END_VAR
// Schreibe Log in regelmässigen Zeitabständen
log_timer( IN := NOT log_timer.Q, PT := sample_rate );
IF log_timer.Q THEN
	triggered := TRUE;
	trigger(clock);
ELSE
	triggered := FALSE;
END_IF

write( data_collector, stack, file_writer_connected );
END_METHOD

END_FUNCTION_BLOCK

// Log/Interfaces/ITF_LogExtension
INTERFACE ITF_LogExtension EXTENDS ITF_Loggable

METHOD getLogTrigger : BOOL
VAR_INPUT
	mode : UINT;
END_VAR
END_METHOD

END_INTERFACE

// Log/Interfaces/ITF_Recordable
INTERFACE ITF_Recordable EXTENDS ITF_Loggable

METHOD enableSelectionMode : BOOL  // returns TRUE if at least one log element is selected.
VAR_INPUT
	enable : BOOL;
END_VAR
END_METHOD

END_INTERFACE

// Log/LogStack/FB_ResponseStackManager
{attribute 'analysis' := '-2'} // yes this is empty
FUNCTION_BLOCK FB_ResponseStackManager
VAR
	response_stack : ARRAY[0..PL_Log.log_stack_size-1] OF ST_ResponseStack;
	log_stack_sent, log_stack_received : ARRAY[0..PL_Log.log_stack_size-1] OF BOOL;
	response_stack_full : BOOL;
END_VAR

METHOD getResponse : ST_ResponseStack
VAR_INPUT
	key : INT;
END_VAR
VAR
	first : INT;
	search : INT;
END_VAR
// Lese Antwort aus response stack

// Finde Eintrag mit gleichem Key im Response Stack
// Der Eintrag befindet sich ungefähr hier.
IF key < PL_Log.log_stack_size THEN
	search := first := key;
ELSE
	search := first := ((key MOD PL_Log.log_stack_size) + 20) MOD PL_Log.log_stack_size;
END_IF

// Suche nächsten Eintrag mit passendem Key
// Der nächste Eintrag ist garantiert der neuste!
WHILE response_stack[search].key <> key DO
	search := (search + 1) MOD PL_Log.log_stack_size;
	IF search = first THEN
		// Response nicht im Stack gefunden.
		RETURN;
	END_IF
END_WHILE

// Eintrag gefunden. Zurückgeben:
getResponse.key := response_stack[search].key;
getResponse.error := response_stack[search].error;
getResponse.fault_code := response_stack[search].fault_code;
log_stack_received[search] := log_stack_sent[search]; // als erledigt markieren.

// Restliche Slots mit diesem Key ebenfalls wieder freigeben.
REPEAT
	search := (search + 1)  MOD PL_Log.log_stack_size;
	IF response_stack[search].key = key THEN
		log_stack_received[search] := log_stack_sent[search];
	END_IF
UNTIL search = first
END_REPEAT;
END_METHOD

METHOD storeResponse : BOOL
VAR_INPUT
	key			: INT;
	error		: BOOL;
	fault_code	: INT;
END_VAR
VAR
	first : INT;
	search	: INT;
END_VAR
// Schreibe Antwort in response stack

// Finde freien Slot oder Eintrag mit gleichem Key im Response Stack
// Um Einträge schneller zu finden, stehen sie immer an der gleichen Stelle.
IF key < PL_Log.log_stack_size THEN
	search := first := key;
ELSE
	search := first := ((key MOD PL_Log.log_stack_size) + 20) MOD PL_Log.log_stack_size;
END_IF

// Falls key nicht an erwarteter stelle ist, weitersuchen, oder den nächsten freien Slot nehmen.
WHILE response_stack[search].key <> key AND log_stack_sent[search] = log_stack_received[search] DO
	search := (search + 1) MOD PL_Log.log_stack_size;
	IF search = first THEN
		// Response Stack ist voll
		response_stack_full := TRUE;
		RETURN;
	END_IF
END_WHILE

response_stack_full := FALSE; // Zurücksetzen.

// Schreibe in Response Stack
response_stack[search].key := key;
response_stack[search].error := error;
response_stack[search].fault_code := fault_code;
log_stack_sent[search] := NOT log_stack_received[search];
END_METHOD

END_FUNCTION_BLOCK

// Math/F_NotZero
FUNCTION F_NotZero : REAL
VAR_INPUT
	maybe_zero : REAL;
END_VAR
VAR
	non_zero_real : REAL := 1E-9;
END_VAR

IF maybe_zero = 0 THEN
	F_NotZero := non_zero_real;
ELSE
	F_NotZero := maybe_zero;
END_IF

END_FUNCTION

// Math/F_Ramp
FUNCTION F_Ramp : REAL
VAR_INPUT
	current : REAL;
	goal	: REAL;
	speed	: REAL;
END_VAR
VAR
END_VAR

F_Ramp := current + LIMIT( -speed, goal - current, speed );

END_FUNCTION

// Mixin/Fallible/ITF_Fallible
INTERFACE ITF_Fallible EXTENDS __SYSTEM.IQueryInterface

PROPERTY get_name : STRING
GET
END_GET
END_PROPERTY

PROPERTY has_error : BOOL
GET
END_GET
END_PROPERTY

END_INTERFACE

// Mixin/Pressure/FB_PressureMixin
FUNCTION_BLOCK FB_PressureMixin
VAR_INPUT
	pressure_unit : E_PressureUnit;
END_VAR

METHOD bar : REAL  // in Bar
VAR_INPUT
	value : REAL;
END_VAR
IF pressure_unit = E_PressureUnit.bar THEN
	bar := value;
ELSIF pressure_unit = E_PressureUnit.pa THEN
	bar := value / 1E5;
ELSE
	bar := value / 1000;
END_IF
END_METHOD

PROPERTY display_accuracy : UINT
GET
// meaningful display accuracy
IF pressure_unit = E_PressureUnit.bar OR pressure_unit = E_PressureUnit.pa THEN
	// for bar
	display_accuracy := 3;
ELSE
	// for mbar
	display_accuracy := 0;
END_IF
END_GET
END_PROPERTY

METHOD from_mbar : REAL
VAR_INPUT
	value : REAL;
END_VAR
IF pressure_unit = E_PressureUnit.bar THEN
	from_mbar := value / 1000;
ELSIF pressure_unit = E_PressureUnit.mbar THEN
	from_mbar := value;
ELSE
	from_mbar := value * 1E2;
END_IF
END_METHOD

METHOD mbar : REAL
VAR_INPUT
	value : REAL;
END_VAR
IF pressure_unit = E_PressureUnit.bar THEN
	mbar := value * 1000;
ELSIF pressure_unit = E_PressureUnit.mbar THEN
	mbar := value;
ELSE
	mbar := value / 1E2;
END_IF
END_METHOD

METHOD pa : REAL
VAR_INPUT
	value : REAL;
END_VAR
IF pressure_unit = E_PressureUnit.bar THEN
	pa := value * 1E5;
ELSIF pressure_unit = E_PressureUnit.mbar THEN
	pa := value * 1E2;
ELSE
	pa := value;
END_IF
END_METHOD

END_FUNCTION_BLOCK

// Physics/SteamCondition/F_P_SAT
FUNCTION F_P_SAT : REAL
// Diese Funktion berechnet der Sättigungsdampfdruck bei einer bestimmten Temperatur
VAR_INPUT
	T : REAL; // Istwert Temperatur
END_VAR
VAR
	i : DINT;	// Array Index
END_VAR
VAR CONSTANT
	// Dieser Array beinhaltet der Sättigungsdampfdruck für Temperaturen von 0..100°C
	// Source: de.wikibooks.org/wiki/Tabellensammlung_Chemie/_Stoffdaten_Wasser
	i_max		: INT := 100;
	sat_press	: ARRAY[ 0..i_max] OF REAL := [6.112, 	6.571,	7.059,	7.580,	8.135,	8.725,	9.352,	10.019,	10.728,	11.481,	12.279,	 13.127,	 14.025,	 14.977,	15.986,	  17.053,	  18.183,	   19.378,	   20.641,	   21.976,	   23.385,	   24.874,		26.444,	 28.101,	 29.847,	   31.687,	  33.626,	35.667,	  37.815,	   40.075,	   42.452,	   44.950,	   47.575,	   50.332, 	   53.227, 	   56.265, 	   59.451, 	   62.793, 	   66.296, 	   69.968, 	   73.813, 	   77.832, 	   82.054, 	   86.463, 	   91.076, 	   95.898, 	   100.939, 	106.206,	   111.708, 	  117.452,	   123.448,	129.074, 136.23, 143.036 , 150.130, 157.523, 165.224, 173.245, 181.596, 190.287, 199.331, 208.738, 218.520, 228.689, 239.257, 250.237, 261.642, 273.485,285.778, 298.536, 311.773, 325.503, 339.740, 354.500, 369.796, 385.646, 402.064, 419.067, 436.671, 454.892, 473.749, 493.257, 513.435, 534.3, 555.871, 578.167, 601.207, 625.009, 649.594, 674.981, 701.190, 728.243, 756.161, 784.964, 814.674, 845.314, 876.906, 909.472, 943.036, 977.620, 1013.25] ;
	delta_T		: REAL:=1.0; // Die Sat.Press-Werte im Array sind für 0, 1, 2,3..100°C angegeben-> deswegen Delta_T := 1
END_VAR

i := TRUNC(	MAX( 0, MIN( i_max-1, T	) )	);
// TRUNC schneidet dem REAL Wert die Kommastellen ab und gibt einen INT zurück: Bsp: TRUNC(1.999) := 1, TRUNC(-1.4) := -1. Zudem muss beachtet
// werden, dass fT im Array-Range bleibt -> deswegen MIN, MAX Bedingungen

F_P_SAT :=  ( T - DINT_TO_REAL(i) ) / delta_T * ( sat_press[ i+1] - sat_press[ i ] ) + sat_press[i];

END_FUNCTION

// Physics/SteamCondition/F_T_SAT
FUNCTION F_T_SAT : REAL
// Diese Funktion berechnet die Sättigungsdampftemperatur bei einem bestimmten Druck
VAR_INPUT
	p : REAL; // Istwert Druck [mbar]
END_VAR
VAR
	i : DINT; // Array Index
END_VAR
VAR CONSTANT
	// Dieser Array beinhaltet der Sättigungsdampfdruck für Temperaturen von 0..110°C
	// Source: de.wikibooks.org/wiki/Tabellensammlung_Chemie/_Stoffdaten_Wasser / Ab 100 bis 110°C : http://webbook.nist.gov/chemistry/fluid/
	i_max		: INT := 110;
	sat_press	: ARRAY[ 0..i_max] OF REAL := [6.112, 	6.571,	7.059,	7.580,	8.135,	8.725,	9.352,	10.019,	10.728,	11.481,	12.279,	 13.127,	 14.025,	 14.977,	15.986,	  17.053,	  18.183,	   19.378,	   20.641,	   21.976,	   23.385,	   24.874,		26.444,	 28.101,	 29.847,	   31.687,	  33.626,	35.667,	  37.815,	   40.075,	   42.452,	   44.950,	   47.575,	   50.332, 	   53.227, 	   56.265, 	   59.451, 	   62.793, 	   66.296, 	   69.968, 	   73.813, 	   77.832, 	   82.054, 	   86.463, 	   91.076, 	   95.898, 	   100.939, 	106.206,	   111.708, 	  117.452,	   123.448,	129.074, 136.23, 143.036 , 150.130, 157.523, 165.224, 173.245, 181.596, 190.287, 199.331, 208.738, 218.520, 228.689, 239.257, 250.237, 261.642, 273.485,285.778, 298.536, 311.773, 325.503, 339.740, 354.500, 369.796, 385.646, 402.064, 419.067, 436.671, 454.892, 473.749, 493.257, 513.435, 534.3, 555.871, 578.167, 601.207, 625.009, 649.594, 674.981, 701.190, 728.243, 756.161, 784.964, 814.674, 845.314, 876.906, 909.472, 943.036, 977.620, 1013.25, 1051.3, 1089.1, 1128.1, 1168.2, 1209.4, 1251.9, 1295.6, 1340.5, 1386.8, 1434.3] ;
	delta_T		: REAL:=1.0; // Die Sat.Temp-Werte im Array sind für 0, 1, 2,3..100°C angegeben-> deswegen Delta_T := 1
END_VAR

i := 0;
WHILE i < i_max AND sat_press[i] < p DO
	i := i+1;
END_WHILE

IF i <= 0 THEN
	F_T_sat := 0.0;
ELSIF (0 < i) AND (i < i_max) THEN
	F_T_sat := (p - sat_press[i-1]) / (sat_press[i] - sat_press[i-1]) * delta_T + DINT_TO_REAL(i-1);
ELSE // i >= iMax
	F_T_sat := INT_TO_REAL(i_max) * delta_T;
END_IF

END_FUNCTION

// Physics/F_sim_pressureFlow
FUNCTION F_sim_pressureFlow : REAL
// Simuliert die änderung des Drucks anhand eines benachbarten drucks
VAR_INPUT
	pressure_this	: REAL;
	volume_this		: REAL;
	pressure_other	: REAL;
	volume_other	: REAL;
	speed			: REAL := 2; // Geschwindigkeit des Druckausgleichs
END_VAR
VAR
END_VAR

F_sim_pressureFlow := F_Ramp(
	current := pressure_this,
	goal	:= ( pressure_this * volume_this + pressure_other * volume_other ) / ( volume_this + volume_other ),
	speed	:= speed * volume_other / ( volume_this + volume_other ) * ABS( pressure_this - pressure_other )/100
);

END_FUNCTION

// TEST/lib/FB_Test
FUNCTION_BLOCK FB_Test
VAR_INPUT
END_VAR
VAR_OUTPUT
	// States
	result : BOOL;
END_VAR
VAR
	// Properties
	name : STRING;
END_VAR

METHOD check : BOOL
VAR_INPUT
	condition : BOOL;
END_VAR
result := condition;
END_METHOD

END_FUNCTION_BLOCK

// TEST/lib/TEST_TEMPLATE
PROGRAM TEST_TEMPLATE
VAR_INPUT
END_VAR
VAR_OUTPUT
	summary : BOOL;
END_VAR
VAR
	//////////
	// Setup
	//


	//////////
	// Process
	stage : UINT;
	i : UINT;

	//////////
	// Results
	tests : ARRAY[0..num_tests] OF FB_Test := [
		( name := 'Test1' )
	];
END_VAR
VAR CONSTANT
	num_tests : UINT := 1;
END_VAR

CASE stage OF
	0: // Reset Tests

		// process
		stage := stage + 1;

	1: // Setup
		//

		// process
		stage := stage + 1;

	2: // Execute
		//

		// process
		stage := stage + 1;

	3: // Check
		//

		// process
		stage := stage + 1;

	4: // Create Summary
		summary := TRUE;
		FOR i := 0 TO num_tests DO
			summary := summary AND tests[i].result;
		END_FOR

		// process
		stage := stage + 1;

	5: // Done

END_CASE

END_PROGRAM

// TEST/Utils/TEST_BITS
PROGRAM TEST_BITS
VAR
	test : ARRAY[0..3] OF BYTE;
END_VAR

// should yield a 5 in test[2]
SET_BIT_IN_BYTE_ARRAY(test, 16, TRUE);
SET_BIT_IN_BYTE_ARRAY(test, 17, TRUE);
SET_BIT_IN_BYTE_ARRAY(test, 18, TRUE);
SET_BIT_IN_BYTE_ARRAY(test, 17, FALSE);

END_PROGRAM

// TEST/TEST
PROGRAM TEST

TEST_TIMESTRUCT_INCREMENT();
TEST_BITS();

END_PROGRAM

// TEST/Utils/TEST_TIMESTRUCT_INCREMENT
PROGRAM TEST_TIMESTRUCT_INCREMENT
VAR_INPUT
END_VAR
VAR_OUTPUT
	summary : BOOL;
END_VAR
VAR
	//////////
	// Setup
	//
	test1 : TIMESTRUCT;
	test2 : TIMESTRUCT;
	test3 : TIMESTRUCT;

	//////////
	// Process
	stage : UINT;
	i : UINT;

	//////////
	// Results
	tests : ARRAY[0..num_tests] OF FB_Test := [
		( name := 'Test1' )
	];
END_VAR
VAR CONSTANT
	num_tests : UINT := 2;

	base1 : TIMESTRUCT := ( wYear := 2019, wMonth := 7, wDay := 23, wHour := 10, wMinute := 23, wSecond := 1, wMilliseconds := 200 );
	base2 : TIMESTRUCT := ( wYear := 2019, wMonth := 7, wDay := 23, wHour := 10, wMinute := 23, wSecond := 1, wMilliseconds := 800 );
	result1 : TIMESTRUCT := ( wYear := 2019, wMonth := 7, wDay := 23, wHour := 10, wMinute := 23, wSecond := 1, wMilliseconds := 700 );
	result2 : TIMESTRUCT := ( wYear := 2019, wMonth := 7, wDay := 23, wHour := 10, wMinute := 23, wSecond := 2, wMilliseconds := 700 );
	result3 : TIMESTRUCT := ( wYear := 2019, wMonth := 7, wDay := 23, wHour := 10, wMinute := 23, wSecond := 2, wMilliseconds := 300 );
END_VAR

CASE stage OF
	0: // Reset Tests
		// process
		stage := stage + 1;

	1: // Setup
		//
		test1 := base1;
		test2 := base1;
		test3 := base2;
		// process
		stage := stage + 1;

	2: // Execute
		//
		test1 := TIMESTRUCT_INCREMENT(test1, 500);
		test2 := TIMESTRUCT_INCREMENT(test2, 1500);
		test3 := TIMESTRUCT_INCREMENT(test3, 500);
		// process
		stage := stage + 1;

	3: // Check
		//
		tests[0].check( assertEqual(test1, result1) );
		tests[1].check( assertEqual(test2, result2) );
		tests[2].check( assertEqual(test3, result3) );
		// process
		stage := stage + 1;

	4: // Create Summary
		summary := TRUE;
		FOR i := 0 TO num_tests DO
			summary := summary AND tests[i].result;
		END_FOR

		// process
		stage := stage + 1;

	5: // Done

END_CASE

METHOD PRIVATE assertEqual : BOOL
VAR_INPUT
	t1 : TIMESTRUCT;
	t2 : TIMESTRUCT;
END_VAR
assertEqual :=
	t1.wYear = t2.wYear
	AND t1.wMonth = t2.wMonth
	AND t1.wDay = t2.wDay
	AND t1.wHour = t2.wHour
	AND t1.wMinute = t2.wMinute
	AND t1.wSecond = t2.wSecond
	AND t1.wMilliseconds = t2.wMilliseconds
;
END_METHOD

END_PROGRAM

// Utils/Bits/SET_BIT_IN_BYTE_ARRAY
FUNCTION SET_BIT_IN_BYTE_ARRAY : BOOL
VAR_IN_OUT
	base : ARRAY[*] OF BYTE;
END_VAR
VAR_INPUT
	index : UINT;
	new_value : BOOL;
END_VAR
VAR
	i : UINT;
END_VAR

i := index / 8;
IF i <= UPPER_BOUND(base, 1) - LOWER_BOUND(base, 1) THEN
	SET_BIT_IN_BYTE_ARRAY := SET_BIT_IN_BYTE(base[i+LOWER_BOUND(base, 1)], index - i*8, new_value);
END_IF

END_FUNCTION

// Utils/Bits/SET_BIT_IN_BYTE
FUNCTION SET_BIT_IN_BYTE : BOOL
VAR_IN_OUT
	base : BYTE;
END_VAR
VAR_INPUT
	index : UINT;
	new_value : BOOL;
END_VAR

SET_BIT_IN_BYTE := TRUE;  //assume success unless it fails
CASE index OF
	0: base.0 := new_value;
	1: base.1 := new_value;
	2: base.2 := new_value;
	3: base.3 := new_value;
	4: base.4 := new_value;
	5: base.5 := new_value;
	6: base.6 := new_value;
	7: base.7 := new_value;
ELSE
	SET_BIT_IN_BYTE := FALSE;  // index out of range
END_CASE

END_FUNCTION

// Utils/Endian/F_IntSwapEndian
FUNCTION F_IntSwapEndian : INT
VAR_INPUT
	value : INT;
END_VAR
VAR
	source : Int16;
	target : Int16;
END_VAR

source.integer := value;
target.bytes[0] := source.bytes[1];
target.bytes[1] := source.bytes[0];
F_IntSwapEndian := target.integer;

END_FUNCTION

// Utils/Endian/F_SafeRealSwapEndian
FUNCTION F_SafeRealSwapEndian : REAL
VAR_INPUT
	source : Float32;
	default : REAL;
END_VAR
VAR
	target : Float32;
	i : UINT;
END_VAR

FOR i := 0 TO 3 DO
	target.bytes[i] := source.bytes[3-i];
END_FOR

IF IsFinite( F_REAL( target.float )) THEN
	F_SafeRealSwapEndian := target.float;
ELSE
	F_SafeRealSwapEndian := default;
END_IF

END_FUNCTION

// Utils/Endian/F_SafeRealSwapWords
FUNCTION F_SafeRealSwapWords : REAL
VAR_INPUT
	source : Float32;
	default : REAL;
END_VAR
VAR
	target : Float32;
	i : UINT;
END_VAR


target.words[0] := source.words[1];
target.words[1] := source.words[0];

IF IsFinite( F_REAL( target.float )) THEN
	F_SafeRealSwapWords := target.float;
ELSE
	F_SafeRealSwapWords := default;
END_IF

END_FUNCTION

// Utils/String/Concat/CONCAT4
FUNCTION CONCAT4 : T_MaxString
VAR_INPUT
	string1 : T_MaxString;
	string2 : T_MaxString;
	string3 : T_MaxString;
	string4 : T_MaxString;
END_VAR
VAR
END_VAR

CONCAT4 := CONCAT( CONCAT ( CONCAT ( string1, string2 ), string3) , string4 );

END_FUNCTION

// Utils/String/Concat/CONCAT6
FUNCTION CONCAT6 : T_MaxString
VAR_INPUT
	string1 : T_MaxString;
	string2 : T_MaxString;
	string3 : T_MaxString;
	string4 : T_MaxString;
	string5 : T_MaxString;
	string6 : T_MaxString;
END_VAR
VAR
END_VAR

CONCAT6 := CONCAT( CONCAT( CONCAT( CONCAT ( CONCAT ( string1, string2 ), string3) , string4 ), string5 ), string6 );

END_FUNCTION

// Utils/String/Placeholder/F_ResolvePlaceholder
FUNCTION F_ResolvePlaceholder : T_MaxString
// Replaces the expression "{placeholder}" in str by "replacement" and returns the result.
// If no placeholder is found, the string is returned unchanged.
VAR_IN_OUT CONSTANT
	str : T_MaxString;
	placeholder : PLACEHOLDER_STRING;
	replacement : T_MaxString;
END_VAR
VAR_OUTPUT
	found : BOOL;
END_VAR

F_ResolvePlaceholder := F_FindAndReplace( str, CONCAT3('{', placeholder, '}'), replacement, found => found );

END_FUNCTION

// Utils/String/F_FindAndReplaceAll
FUNCTION F_FindAndReplaceAll : STRING
VAR_INPUT
	str : T_MaxString;
	find_str : T_MaxString;
	replace_str : T_MaxString;
END_VAR
VAR
	found : BOOL;
END_VAR

REPEAT
	str := F_FindAndReplace(str, find_str, replace_str, found => found);
UNTIL NOT found
END_REPEAT;
F_FindAndReplaceAll := str;

END_FUNCTION

// Utils/String/F_Glue
FUNCTION F_Glue : T_MaxString
// concats pre and post with glue if both are non-empty
// if pre or post are empty, returns the non-empty one
VAR_INPUT
	pre : T_MaxString;
	glue : T_MaxString;
	post : T_MaxString;
END_VAR

IF pre <> '' AND post <> '' THEN
	F_Glue := CONCAT3( pre, glue, post );
ELSE
	F_Glue := CONCAT( pre, post );
END_IF

END_FUNCTION

// Utils/String/F_ReplaceX
FUNCTION F_ReplaceX : T_MaxString
// Ersetzt den Ausdruck "{X}" in str durch insert.
// Wenn kein {X} gefunden wird, wird str unverändert zurückgegeben
VAR_INPUT
	str	: T_MaxString;
	insert : STRING;
END_VAR

F_ReplaceX := F_FindAndReplace( str, '{X}', insert );

END_FUNCTION

// Utils/String/FILL_WIDTH
FUNCTION FILL_WIDTH : STRING[max_size]
// Füllt einen String in von Links mit einem zeichen fill bis zur Länge width auf.
VAR_INPUT
	in : STRING[max_size];
	width : INT;
	fill : STRING[1];
END_VAR
VAR CONSTANT
	max_size : INT := 40;
END_VAR

FILL_WIDTH := in;
width := MIN( MIN( width, max_size ), 255 );

WHILE LEN(FILL_WIDTH) < width DO
	FILL_WIDTH := CONCAT(fill, FILL_WIDTH);
END_WHILE

END_FUNCTION

// Utils/Ternary/BOOL_TO_TERNARY
FUNCTION BOOL_TO_TERNARY : E_Ternary
VAR_INPUT
	value : BOOL;
END_VAR

IF value THEN
	BOOL_TO_TERNARY := E_Ternary.yes;
ELSE
	BOOL_TO_TERNARY := E_Ternary.no;
END_IF

END_FUNCTION

// Utils/Time/FB_Blinker
FUNCTION_BLOCK FB_Blinker
VAR_INPUT
	start			: BOOL;
	on_duration		: TIME;
	off_duration 	: TIME;
END_VAR
VAR_OUTPUT
	q 				: BOOL;
END_VAR
VAR
	ton_1			: TON;
	ton_2			: TON;
END_VAR

// Blinktakt mit Hilfe von 2 Timern
// ON
ton_1(
	IN := start AND NOT ton_2.Q,
	PT := on_duration,
	Q=> q
);
// OFF
ton_2(
	IN := ton_1.Q,
	PT := off_duration
);

END_FUNCTION_BLOCK

// Utils/Time/FB_TimeDelta
FUNCTION_BLOCK FB_TimeDelta
// Bestimmt die Zeitdifferenz zwischen Aufrufen mit bis zu 429.4967295s differenz.
VAR_INPUT
END_VAR
VAR_OUTPUT
	delta 		: LREAL; 	// Zeitdifferenz seit letztem Aufruf dieses FBs [s]
	ready		: BOOL;		// TRUE, dieser FB bereit ist und sinnvolle Werte liefert.
END_VAR
VAR
	timer_now 	: GETCPUCOUNTER;
	timer_last 	: UDINT;
	init		: BOOL;
END_VAR

// Zeitdifferenz zum letzen Aufruf berechnen
timer_now();
delta := UDINT_TO_LREAL( timer_now.cpuCntLoDW - timer_last )/1E7; // [100ns] underflow wird korrekt gehandhabt
timer_last := timer_now.cpuCntLoDW;
// Dieser Funktionsblock liefert erst beim zweiten Aufruf einen sinnvollen wert.
ready := init;
init := TRUE;

IF NOT ready THEN
	delta := 0; // beim ersten mal 0 statt bedeutungslosen wert zurückgeben.
END_IF

METHOD reset : BOOL
// FB zurücksetzen. Dies sollte immer gemacht werden, wenn FB für grossen Zeitinterwall nicht mehr genutzt wird.
VAR_INPUT
END_VAR
init 	:= FALSE;
ready 	:= FALSE;
END_METHOD

END_FUNCTION_BLOCK

// Utils/Time/FB_TON_PAUSABLE
FUNCTION_BLOCK FB_TON_PAUSABLE
VAR_INPUT
	IN		: BOOL;
	PT		: TIME;
	PAUSE	: BOOL;
END_VAR
VAR_OUTPUT
	Q		: BOOL;
	ET		: TIME;
	PAUSED	: BOOL; // könnte man auch mit einem VAR_IN_OUT lösen. Nachteil würde bei Funktionsaufrufe immer PAUSE verlangen.
END_VAR
VAR
	rtPause 	: R_TRIG;	// steigende Flanke (Rising Edge)
	ElapsedTime	: TIME;		// Zwischenspeicher der bereits vergangene Zeit
	ton			: TON;
END_VAR

// reset Time Zwischenspeicher
IF NOT IN THEN
	ElapsedTime := T#0S;
END_IF

PAUSED := PAUSE;

// run Flankenerkennung
rtPause(CLK := PAUSE);

// update Zwischenspeicher, wenn Pause auslöst
IF rtPause.Q THEN
	ElapsedTime := ElapsedTime + ton.ET;
END_IF

// run TON
ton(IN := IN AND NOT PAUSE, PT := PT - ElapsedTime);

// Outputs
Q := ton.Q;
ET := ElapsedTime + ton.ET;

END_FUNCTION_BLOCK

// Utils/Time/TIME_TO_FSTRING
FUNCTION TIME_TO_FSTRING : STRING
// Formatiert eine Dauer in ein Menschenfreundliches Format für die Visu.
VAR_INPUT
	t : TIME := T#3D;
	low_unit : E_TIME_UNIT;
	high_unit : E_TIME_UNIT;
END_VAR
VAR
	cur, next : UDINT;
	unit : INT;
	factor : ARRAY[ E_TIME_UNIT.millisecond..E_TIME_UNIT.day ] OF UINT := [ 1000, 60, 60, 24, 1 ];
	delimiter : ARRAY[ E_TIME_UNIT.millisecond..E_TIME_UNIT.day ] OF STRING[6] := [ '.', ':', ':', ' Tage ', '' ];
	width : ARRAY[ E_TIME_UNIT.millisecond..E_TIME_UNIT.day ] OF INT := [ 4, 2, 2, 1, 1 ];
END_VAR

next := TIME_TO_UDINT(t);

FOR unit := E_TIME_UNIT.millisecond TO E_TIME_UNIT.day DO
	IF high_unit > unit THEN
		cur := next MOD factor[unit];
		next := (next - cur)/factor[unit];
	ELSE
		cur := next;
	END_IF
	IF low_unit <= unit THEN
		IF high_unit > unit AND next <> 0 THEN
			TIME_TO_FSTRING := CONCAT( FILL_WIDTH( UDINT_TO_STRING( cur ), width[unit], '0' ), TIME_TO_FSTRING);
			TIME_TO_FSTRING := CONCAT( delimiter[unit], TIME_TO_FSTRING );
		ELSE
			TIME_TO_FSTRING := CONCAT( UDINT_TO_STRING( cur ), TIME_TO_FSTRING);
			EXIT;
		END_IF
	END_IF
END_FOR

// Suffix
CASE unit OF
	E_TIME_UNIT.millisecond:
		TIME_TO_FSTRING := CONCAT( TIME_TO_FSTRING, ' ms' );

	E_TIME_UNIT.second:
		TIME_TO_FSTRING := CONCAT( TIME_TO_FSTRING, ' s' );
END_CASE

END_FUNCTION

// Utils/FB_RememberRestore
FUNCTION_BLOCK FB_RememberRestore
// Merkt sich einen Wert.
VAR_INPUT
END_VAR
VAR_OUTPUT
	stored : BOOL; // TRUE, wenn ein Wert gemerkt ist.
END_VAR
VAR
	memory : BOOL; // Wert der Gemerkt werden soll
END_VAR

METHOD remember : BOOL
// Bei mehrfachem aufruf von remember wird der gemerkte Wert nicht überschrieben
// Erst wenn wieder "restored" wurde, kann neu "remembered" werden
VAR_INPUT
	value : BOOL;
END_VAR
IF NOT stored THEN
	memory := value;
	stored := TRUE;
END_IF
END_METHOD

METHOD restore : BOOL
// Gibt den Merker wieder frei.
// Bei mehrfachem Aufruf wird der zuletzt gemerkte Wert weiterhin zurückgegeben.
VAR_INPUT
END_VAR
stored := FALSE;
restore := memory;
END_METHOD

END_FUNCTION_BLOCK

// Utils/FB_ResourceManager
FUNCTION_BLOCK FB_ResourceManager
VAR_INPUT
END_VAR
VAR_OUTPUT
END_VAR
VAR
	resource_register : ARRAY[1..max_resource_id] OF BOOL;
	num_registered_resources : UINT;
	resource_limit : UINT(0..max_resource_id); // Anzahl resourcen die maximal vergeben werden können.
END_VAR
VAR CONSTANT
	max_resource_id : UINT := 36;
END_VAR

PROPERTY available : UINT
GET
available := resource_limit - num_registered_resources;
END_GET
END_PROPERTY

METHOD FB_init : BOOL
VAR_INPUT
	bInitRetains : BOOL; // if TRUE, the retain variables are initialized (warm start / cold start)
	bInCopyCode  : BOOL;  // if TRUE, the instance afterwards gets moved into the copy code (online change)
	_limit: UINT(0..max_resource_id); // Falls höhere Werte nötig sind, muss maxResourceID erhöht werden.
END_VAR
resource_limit := _limit;
END_METHOD

METHOD release : BOOL
VAR_INPUT
	id : UINT;
END_VAR
IF id > 0 AND id <= max_resource_id AND resource_register[id] = TRUE THEN
	num_registered_resources := num_registered_resources - 1;
	resource_register[id] := FALSE;
END_IF
END_METHOD

METHOD reserve : BOOL
VAR_INPUT
	id : UINT;
END_VAR
IF resource_register[id] = TRUE THEN // Resource bereits reserviert
	reserve := TRUE;
ELSIF id > 0 AND id <= max_resource_id AND resource_register[id] = FALSE // resource ist noch frei und wird reserviert.
	AND num_registered_resources < resource_limit  THEN
		num_registered_resources := num_registered_resources + 1;
		resource_register[id] := TRUE;
		reserve := TRUE;
ELSE // keine freie Resource
	reserve := FALSE;
END_IF
END_METHOD

END_FUNCTION_BLOCK

// i18n/Frame_SwitchLanguage
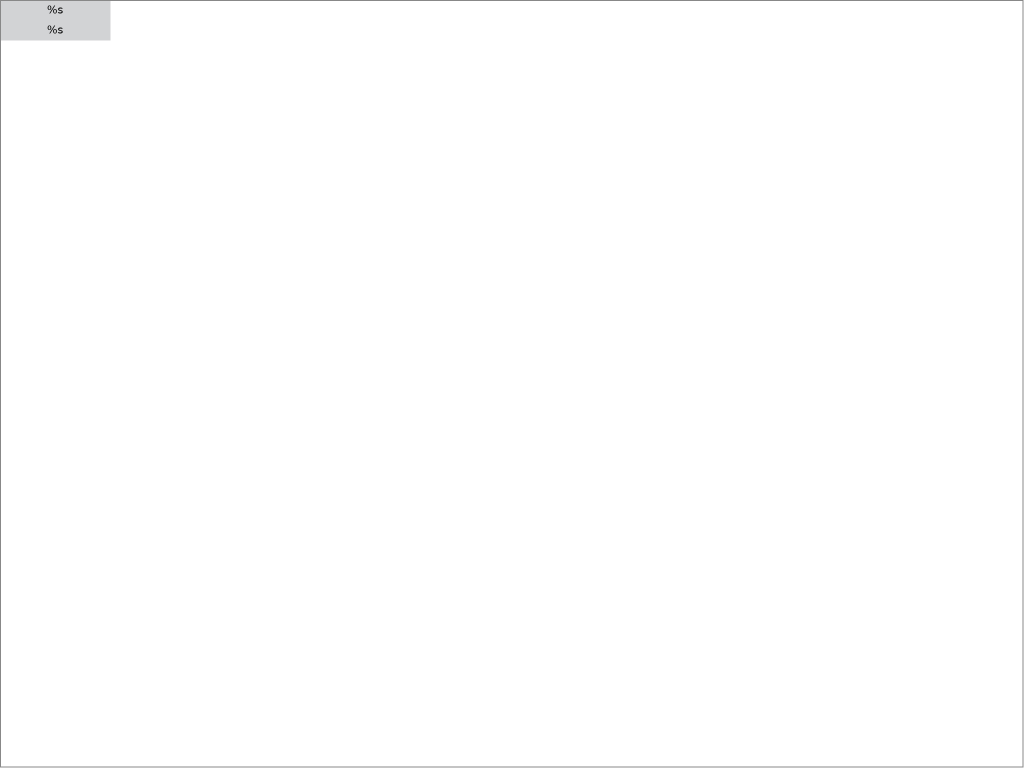
VISUALIZATION Frame_SwitchLanguage  // 1024x768
VAR_IN_OUT
	
END_VAR
VAR CONSTANT
	de : E_Language := E_Language.de;
	en : E_Language := E_Language.en;
END_VAR
    Rectangle (0,0 110x20), "%s", text variable: de
        OnMouseClick:  ChangeLanguage=de
    Rectangle (0,20 110x20), "%s", text variable: en
        OnMouseClick:  ChangeLanguage=en
END_VISUALIZATION

// ManualRecording/Frame_ManualRecording_display
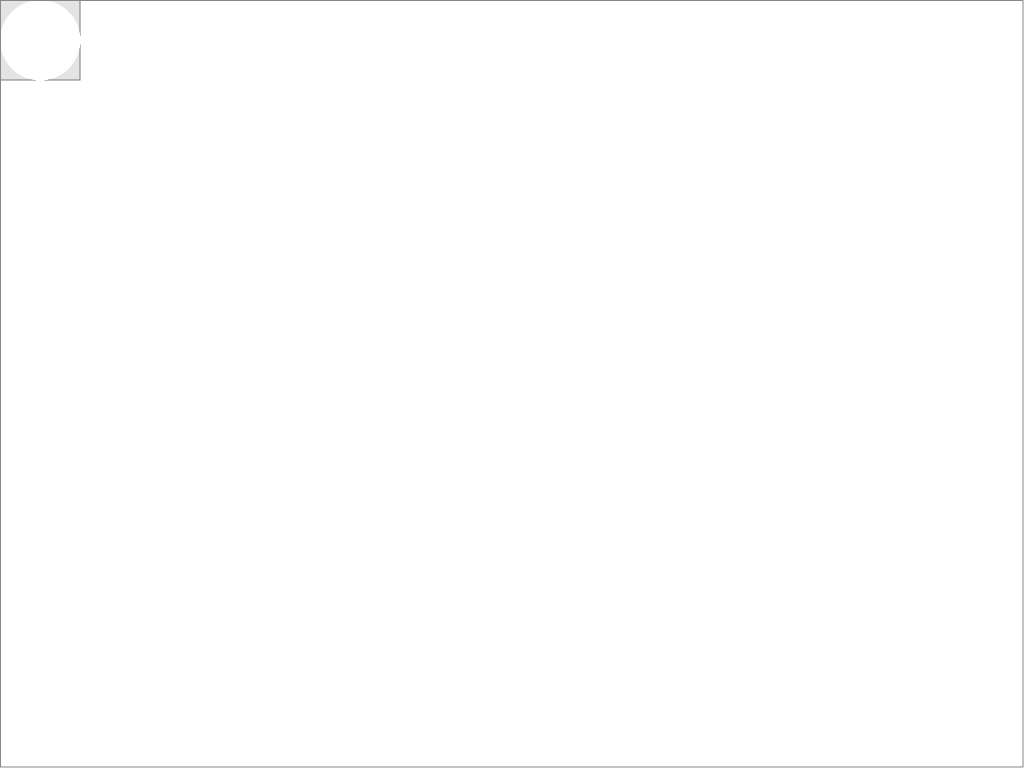
VISUALIZATION Frame_ManualRecording_display  // 1024x768
VAR_IN_OUT
	record : ST_Record;
END_VAR
    PushSwitch (0,0 80x80), variable: record.enabled, invisible if: NOT record.selection_mode AND NOT record.enabled, input disabled if: NOT record.selection_mode, behaviour: TOGGLE, style: Switch-PushSwitch-Red
    Ellipse (0,0 80x80), invisible if: record.selection_mode OR NOT record.enabled
END_VISUALIZATION

// Utils/Limits/Visu/Frame_IntLimits
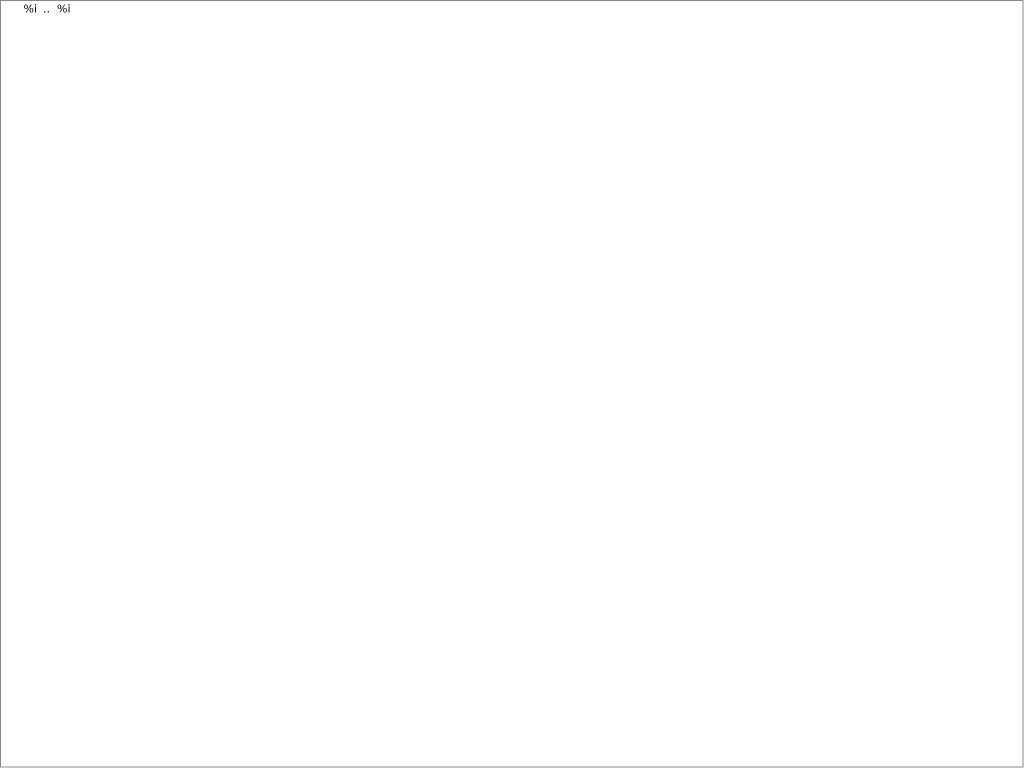
VISUALIZATION Frame_IntLimits  // 1024x768
VAR_IN_OUT
	limits : ST_IntLimits;
END_VAR
    Rectangle (0,0 40x18), "%i", text variable: limits.low
    Rectangle (40,0 11x18), ".."
    Rectangle (54,0 47x18), "%i", text variable: limits.high
END_VISUALIZATION

// Utils/Limits/Visu/Frame_RealLimits
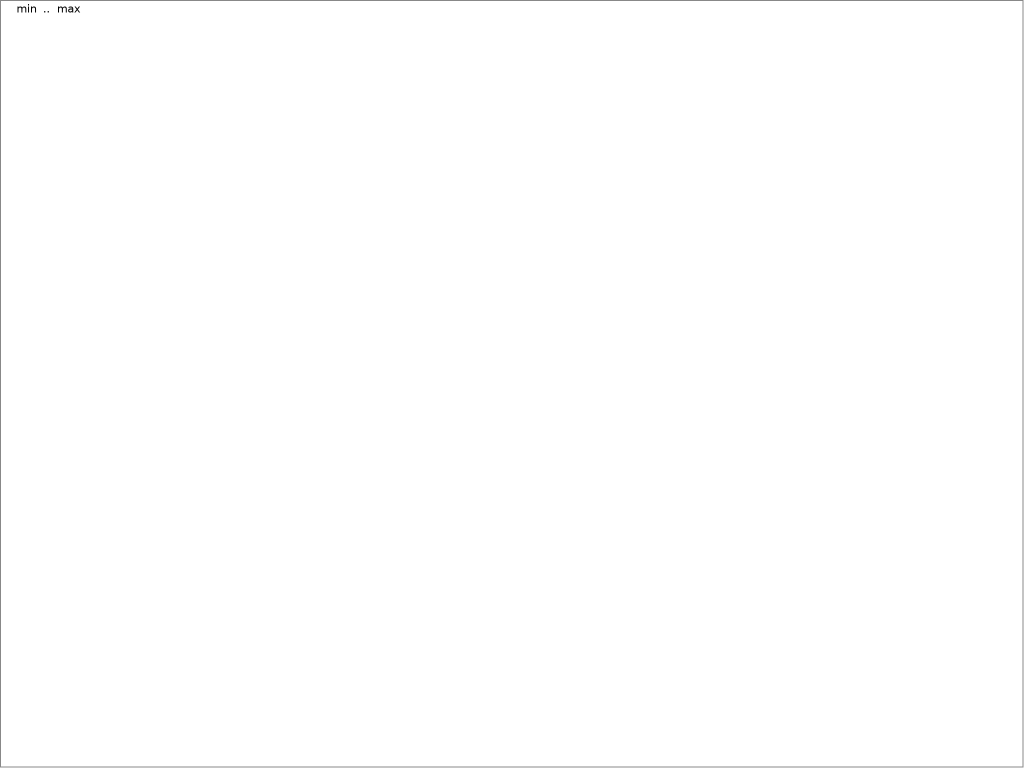
VISUALIZATION Frame_RealLimits  // 1024x768
VAR_IN_OUT
	limits : ST_RealLimits;
END_VAR
    Rectangle (0,0 40x18), "min", text variable: limits.low, text list: 'TL_DisplayAccuracy', text index: limits.display_accuracy
    Rectangle (40,0 11x18), ".."
    Rectangle (54,0 47x18), "max", text variable: limits.high, text list: 'TL_DisplayAccuracy', text index: limits.display_accuracy
END_VISUALIZATION

// Utils/Limits/Visu/Frame_UdintLimits
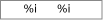
VISUALIZATION Frame_UdintLimits  // 103x20
VAR_IN_OUT
	limits : ST_UdintLimits;
END_VAR
    Rectangle (54,0 47x18), "%i", text variable: limits.high
    Rectangle (0,0 40x18), "%i", text variable: limits.low
END_VISUALIZATION

// Utils/Limits/Visu/Frame_UsintLimits
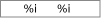
VISUALIZATION Frame_UsintLimits  // 101x18
VAR_IN_OUT
	limits : ST_UsintLimits;
END_VAR
    Rectangle (54,0 47x18), "%i", text variable: limits.high
    Rectangle (0,0 40x18), "%i", text variable: limits.low
END_VISUALIZATION

(* text list TL_DisplayAccuracy (id | default)
  0 | %1.0f
  1 | %1.1f
  2 | %1.2f
  3 | %1.3f
  4 | %1.4f
   |  *)
